# B&R Automation Studio project OpcUaSample410_BrbLibUa103 (part 9)

#### Types.typ - Exported data types
```iecst
(*General*)

TYPE
	BrbErrorUa_ENUM :
		( (*OpcUa-Error-Stati*)
		eBRB_ERR_UA_ERROR := 51000,
		eBRB_ERR_UA_NO_ELEMENTS := 51001,
		eBRB_ERR_UA_INVALID_INDEX := 51002,
		eBRB_ERR_UA_NOT_CONNECTED := 51003,
		eBRB_ERR_UA_NOT_RUNNING := 51004
		);
END_TYPE

(*General - Attributes*)

TYPE
	BrbUaNodeInfoAttribute_TYP : 	STRUCT  (*Attribut-Info*)
		sName : STRING[nBRBUA_ATTRIBUTE_NAME_CHAR_MAX]; (*Name des Attributs*)
		sValue : STRING[nBRBUA_VALUE_TEXT_CHAR_MAX]; (*Wert des Attributs als Text*)
	END_STRUCT;
	BrbUaNodeInfoAttributes_TYP : 	STRUCT  (*Attribute-Liste der Infos*)
		Attribute : ARRAY[0..nBRBUA_ATTRIBUTES_INDEX_MAX]OF BrbUaNodeInfoAttribute_TYP; (*Attribute-Liste der Infos*)
	END_STRUCT;
END_TYPE

(*General - ByteStrings*)
(*General - ServerInfo*)

TYPE
	BrbUaServerNamespacesArray_TYP : 	STRUCT  (*Array für Namespaces*)
		Length : UAArrayLength;
		Data : ARRAY[0..nBRBUA_SRVDIAG_NAMESPACE_IDX_MAX]OF STRING[nBRBUA_NAMESPACE_URI_CHAR_MAX];
	END_STRUCT;
	BrbUaServerBuildInfo_TYP : 	STRUCT  (*Build-Daten des Servers*)
		sProductUri : STRING[255];
		sManufacturerName : STRING[255];
		sProductName : STRING[255];
		sSoftwareVersion : STRING[255];
		sBuildNumber : STRING[255];
		dtBuildDate : DATE_AND_TIME;
	END_STRUCT;
	BrbUaServerState_ENUM :
		( (*Server-Status*)
		eBRBUA_SRVSTATE_RUNNING,
		eBRBUA_SRVSTATE_FAILED,
		eBRBUA_SRVSTATE_NOCONFIG,
		eBRBUA_SRVSTATE_SUSPENDED,
		eBRBUA_SRVSTATE_SHUTDOWN,
		eBRBUA_SRVSTATE_TEST,
		eBRBUA_SRVSTATE_COMMFAULT,
		eBRBUA_SRVSTATE_UNKNOWN
		);
	BrbUaServerStatus_TYP : 	STRUCT  (*Status-Daten des Servers*)
		dtStartTime : DATE_AND_TIME;
		dtCurrentTime : DATE_AND_TIME;
		eServerState : BrbUaServerState_ENUM;
		BuildInfo : BrbUaServerBuildInfo_TYP;
		nSecondsTillShutdown : UDINT;
		ShutdownReason : UALocalizedText;
	END_STRUCT;
END_TYPE

(*General - ServerDiag*)

TYPE
	BrbUaServerDiagData_TYP : 	STRUCT  (*Diagnose-Daten einer Session*)
		nServerViewCount : UDINT;
		nCurrentSessionCount : UDINT;
		nCumulatedSessionCount : UDINT;
		nSecurityRejectedSessionCount : UDINT;
		nRejectedSessionCount : UDINT;
		nSessionTimeoutCount : UDINT;
		nSessionAbortCount : UDINT;
		nCurrentSubscriptionCount : UDINT;
		nCumulatedSubscriptionCount : UDINT;
		nPublishingIntervalCount : UDINT;
		nSecurityRejectedRequestsCount : UDINT;
		nRejectedRequestsCount : UDINT;
	END_STRUCT;
	BrbUaApplicationType_ENUM :
		( (*Applikations-Typen*)
		eBRBUA_APPTYPE_SERVER, (*Nur Server*)
		eBRBUA_APPTYPE_CLIENT, (*Nur Client*)
		eBRBUA_APPTYPE_CLIENT_AND_SERVER, (*Client und Server*)
		eBRBUA_APPTYPE_DISCOVERY_SERVER (*Nur Discovery-Server*)
		);
	BrbUaApplicationDescription_TYP : 	STRUCT  (*Applikations-Beschreibung*)
		sApplicationUri : STRING[255];
		sProductUri : STRING[255];
		ApplicationName : UALocalizedText;
		eApplicationType : BrbUaApplicationType_ENUM;
		sGatewayServerUri : STRING[255];
		sDiscoveryProfileUri : STRING[255];
		DiscoveryUrlsLength : UANoOfElements;
		sDiscoveryUrls : ARRAY[0..9]OF STRING[255];
	END_STRUCT;
	BrbUaServiceCounterData_TYP : 	STRUCT  (*Zähler für Service-Daten*)
		nTotalCount : UDINT;
		nErrorCount : UDINT;
	END_STRUCT;
	BrbUaSessDiagData_TYP : 	STRUCT  (*Diagnose-Daten einer Session*)
		SessionId : UANodeID;
		sSessionName : STRING[255];
		ClientDescription : BrbUaApplicationDescription_TYP;
		sServerUri : STRING[255];
		sEndpointUrl : STRING[255];
		LocaleIdsCount : UANoOfElements;
		sLocaleIds : ARRAY[0..nBRBUA_SRVDIAG_LOCALES_INDEX_MAX]OF STRING[7];
		rActualSessionTimeout : LREAL;
		nMaxResponseMessageSize : UDINT;
		dtClientConnectionTime : DATE_AND_TIME;
		dtClientLastContactTime : DATE_AND_TIME;
		nCurrentSubscriptionsCount : UDINT;
		nCurrentMonitoredItemsCount : UDINT;
		nCurrentPublishRequestsInQueue : UDINT;
		TotalRequestCount : BrbUaServiceCounterData_TYP;
		nUnauthorizedRequestCount : UDINT;
		ReadCount : BrbUaServiceCounterData_TYP;
		HistoryReadCount : BrbUaServiceCounterData_TYP;
		WriteCount : BrbUaServiceCounterData_TYP;
		HistoryUpdateCount : BrbUaServiceCounterData_TYP;
		CallCount : BrbUaServiceCounterData_TYP;
		CreateMonitoredItemsCount : BrbUaServiceCounterData_TYP;
		ModifyMonitoredItemsCount : BrbUaServiceCounterData_TYP;
		SetMonitoringModeCount : BrbUaServiceCounterData_TYP;
		SetTriggeringCount : BrbUaServiceCounterData_TYP;
		DeleteMonitoredItemsCount : BrbUaServiceCounterData_TYP;
		CreateSubscriptionCount : BrbUaServiceCounterData_TYP;
		ModifySubscriptionCount : BrbUaServiceCounterData_TYP;
		SetPublishingModeCount : BrbUaServiceCounterData_TYP;
		PublishCount : BrbUaServiceCounterData_TYP;
		RepublishCount : BrbUaServiceCounterData_TYP;
		TransferSubscriptionsCount : BrbUaServiceCounterData_TYP;
		DeleteSubscriptionsCount : BrbUaServiceCounterData_TYP;
		AddNodesCount : BrbUaServiceCounterData_TYP;
		AddReferencesCount : BrbUaServiceCounterData_TYP;
		DeleteNodesCount : BrbUaServiceCounterData_TYP;
		DeleteReferencesCount : BrbUaServiceCounterData_TYP;
		BrowseCount : BrbUaServiceCounterData_TYP;
		BrowseNextCount : BrbUaServiceCounterData_TYP;
		TranslateBrowsePathToNodeIdCount : BrbUaServiceCounterData_TYP;
		QueryFirstCount : BrbUaServiceCounterData_TYP;
		QueryNextCount : BrbUaServiceCounterData_TYP;
		RegisterNodesCount : BrbUaServiceCounterData_TYP;
		UnregisterNodesCount : BrbUaServiceCounterData_TYP;
	END_STRUCT;
	BrbUaSessDiagArray_TYP : 	STRUCT  (*Array für Session-Diagnose*)
		Length : UAArrayLength;
		Data : ARRAY[0..nBRBUA_SRVDIAG_SESSION_INDEX_MAX]OF BrbUaSessDiagData_TYP;
	END_STRUCT;
	BrbUaMessageSecurityMode_ENUM :
		( (*Message-Secutity-Modes*)
		eBRBUA_SECMODE_INVALID, (*Ungültig*)
		eBRBUA_SECMODE_NONE, (*Keine Security*)
		eBRBUA_SECMODE_SIGN, (*Nur Signierung*)
		eBRBUA_SECMODE_SIGN_AND_ENCRYPT (*Signierung und Verschlüsselung*)
		);
	BrbUaSessSecDiagData_TYP : 	STRUCT  (*Security-Diagnose-Daten einer Session*)
		SessionId : UANodeID;
		sClientUserIdOfSession : STRING[64];
		ClientUserIdHistoryCount : UANoOfElements;
		sClientUserIdHistory : ARRAY[0..nBRBUA_SRVDIAG_USERHIST_IDX_MAX]OF STRING[32];
		sAuthenticationMechanism : STRING[64];
		sEncoding : STRING[64];
		sTransportProtocol : STRING[64];
		eSecurityMode : BrbUaMessageSecurityMode_ENUM;
		sSecurityPolicyUri : STRING[64];
		ClientCertificate : ARRAY[0..nBRBUA_CERT_ARRAY_INDEX_MAX]OF USINT;
	END_STRUCT;
	BrbUaSessSecDiagArray_TYP : 	STRUCT  (*Array für Security-Session-Diagnose*)
		Length : UAArrayLength;
		Data : ARRAY[0..nBRBUA_SRVDIAG_SESSION_INDEX_MAX]OF BrbUaSessSecDiagData_TYP;
	END_STRUCT;
	BrbUaSubscriptDiagData_TYP : 	STRUCT  (*Diagnose-Daten einer Subscription*)
		SessionId : UANodeID;
		nSubscriptionId : UDINT;
		nPriority : USINT;
		rPublishingInterval : LREAL;
		nMaxKeepAliveCount : UDINT;
		nMaxLifetimeCount : UDINT;
		nMaxNotificationsPerPublish : UDINT;
		bPublishingEnabled : BOOL;
		nModifyCount : UDINT;
		nEnableCount : UDINT;
		nDisableCount : UDINT;
		nRepublishRequestCount : UDINT;
		nRepublishMessageRequestCount : UDINT;
		nRepublishMessageCount : UDINT;
		nTransferRequestCount : UDINT;
		nTransferredToAltClientCount : UDINT;
		nTransferredToSameClientCount : UDINT;
		nPublishRequestCount : UDINT;
		nDataChangeNotificationsCount : UDINT;
		nEventNotificationsCount : UDINT;
		nNotificationsCount : UDINT;
		nLatePublishRequestCount : UDINT;
		nCurrentKeepAliveCount : UDINT;
		nCurrentLifetimeCount : UDINT;
		nUnacknowledgedMessageCount : UDINT;
		nDiscardedMessageCount : UDINT;
		nMonitoredItemCount : UDINT;
		nDisabledMonitoredItemCount : UDINT;
		nMonitoringQueueOverflowCount : UDINT;
		nNextSequenceNumber : UDINT;
		nEventQueueOverflowCount : UDINT;
	END_STRUCT;
	BrbUaSubscriptDiagArray_TYP : 	STRUCT  (*Array für Subscription-Diagnose*)
		Length : UAArrayLength;
		Data : ARRAY[0..nBRBUA_SRVDIAG_SUBSCR_INDEX_MAX]OF BrbUaSubscriptDiagData_TYP;
	END_STRUCT;
END_TYPE

(*Client - RunClient*)

TYPE
	UAByteStringBrbEventId_TYP : 	STRUCT  (*EventId als ByteString mit Länge 16*)
		Length : DINT; (*Länge der Daten (sollte mit 16 besetzt werden)*)
		Data : ARRAY[0..nBRBUA_EVENTID_INDEX_MAX]OF USINT; (*Bytes der EventId*)
	END_STRUCT;
	BrbUaRcCfg_TYP : 	STRUCT  (*Verbindungs-Parameter*)
		sCfgDataObjName : STRING[nBRBUA_DATOBJECT_NAME_CHAR_MAX]; (*Name des Datenobjekts*)
		sServerEndpointUrl : STRING[sBRBUA_ENDPOINT_URL_CHAR_MAX]; (*Endpoint-Url*)
		SessionConnectInfo : UASessionConnectInfo; (*Angaben zur Verbindung*)
		tConnectTimeout : TIME; (*Timeout für den Connect in [ms]*)
		tAccessTimeout : TIME; (*Timeout für Zugriff auf den Server in [ms]*)
	END_STRUCT;
	BrbUaRcCommandos_ENUM :
		( (*Client-Kommandos*)
		eBRB_RCCLTCMD_NONE, (*Aktuell kein Kommando*)
		eBRB_RCCLTCMD_CONNECT, (*Verbindung aufbauen*)
		eBRB_RCCLTCMD_DISCONNECT (*Verbindung trennen*)
		);
	BrbUaRcConnection_TYP : 	STRUCT  (*Daten der Verbindung*)
		nConnectionHandle : UDINT; (*Handle der Verbindung*)
		nErrorId : DWORD; (*OpcUa-Fehler beim Verbinden*)
		nConnectTries : UDINT; (*Connect-Versuche*)
		nInterruptedCount : UDINT; (*Anzahl der Verbindungs-Unterbrechungen*)
	END_STRUCT;
	BrbUaRcNamespaces_TYP : 	STRUCT  (*Daten der Namespaces*)
		nNamespaceCount : UINT; (*Anzahl der Namespaces*)
		pNamespaces : {REDUND_UNREPLICABLE} UDINT; (*Interner Zeiger*)
		nMemLen : UDINT; (*Interne Speichergröße*)
	END_STRUCT;
	BrbUaRcNamespace_TYP : 	STRUCT  (*Daten eines Namespaces*)
		sNamespaceUri : STRING[nBRBUA_NAMESPACE_URI_CHAR_MAX]; (*Namespace-Uri aus dem Datenobjekt*)
		nNamespaceIndex : UINT; (*Server-Namespace-Index*)
		nErrorId : DWORD; (*OpcUa-Fehler-Status*)
	END_STRUCT;
	BrbUaRcNodeHandles_TYP : 	STRUCT  (*Daten der NodeHandles*)
		nNodeHandleCount : UINT; (*Anzahl der NodeHandles*)
		pStart : UDINT; (*Interner Zeiger*)
		pDatObjNamespaceIndices : {REDUND_UNREPLICABLE} UDINT; (*Interner Zeiger*)
		pNodeIds : {REDUND_UNREPLICABLE} UDINT; (*Interner Zeiger*)
		pNodeHandleErrorIds : {REDUND_UNREPLICABLE} UDINT; (*Interner Zeiger*)
		pNodeHandles : {REDUND_UNREPLICABLE} UDINT; (*Interner Zeiger*)
		nMemLen : UDINT; (*Interne Speichergröße*)
	END_STRUCT;
	BrbUaRcNodeHandle_TYP : 	STRUCT  (*Daten eines NodeHandles*)
		nDatObjNamespaceIndex : UINT; (*Namespace-Index laut Datenobjekt*)
		NodeId : UANodeID; (*NodeId laut Datenobjekt*)
		nErrorId : DWORD; (*OpcUa-Fehler-Status beim Ermitteln des NodeHandles*)
		nNodeHandle : DWORD; (*Ermittelter NodeHandle*)
	END_STRUCT;
	BrbUaRcReadBlocks_TYP : 	STRUCT  (*Daten der ReadBlocks*)
		nBlockCount : UINT; (*Anzahl der ReadBlocks*)
		pBlocks : {REDUND_UNREPLICABLE} UDINT; (*Interner Zeiger*)
		nMemLen : UDINT; (*Interne Speichergröße*)
	END_STRUCT;
	BrbUaRcReadBlockIntern_TYP : 	STRUCT  (*Interne Daten eines ReadBlocks*)
		nReadItemCount : UINT; (*Anzahl der ReadItems*)
		pRiStart : UDINT; (*Interner Zeiger*)
		pRiDatObjNamespaceIndices : UDINT; (*Interner Zeiger*)
		pRiNodeIds : UDINT; (*Interner Zeiger*)
		pRiNodeAddInfos : UDINT; (*Interner Zeiger*)
		pRiVariables : UDINT; (*Interner Zeiger*)
		pRiNodeErrorIds : UDINT; (*Interner Zeiger*)
		pRiTimestamps : UDINT; (*Interner Zeiger*)
		nMemLen : UDINT; (*Interne Speichergröße*)
	END_STRUCT;
	BrbUaRcReadBlock_TYP : 	STRUCT  (*Daten eines ReadBlocks*)
		nReadItemCount : UINT; (*Anzahl der ReadItems*)
	END_STRUCT;
	BrbUaRcReadItem_TYP : 	STRUCT  (*Daten eines ReadItems*)
		nDatObjNamespaceIndex : UINT; (*Namespace-Index laut Datenobjekt*)
		NodeId : UANodeID; (*NodeId laut Datenobjekt*)
		AddInfo : UANodeAdditionalInfo; (*Zusatzangaben für den Zugriff*)
		sVar : STRING[nBRBUA_VARNAME_TEXT_CHAR_MAX]; (*Name der gemappten Variable*)
		dtTimestamp : DATE_AND_TIME; (*Zeitstempel der letzten Aktion*)
		nErrorId : DWORD; (*OpcUa-Fehler-Status*)
	END_STRUCT;
	BrbUaRcWriteBlocks_TYP : 	STRUCT  (*Daten der WriteBlocks*)
		nBlockCount : UINT; (*Anzahl der WriteBlocks*)
		pBlocks : {REDUND_UNREPLICABLE} UDINT; (*Interner Zeiger*)
		nMemLen : UDINT; (*Interne Speichergröße*)
	END_STRUCT;
	BrbUaRcWriteBlockIntern_TYP : 	STRUCT  (*Interne Daten eines WriteBlocks*)
		nWriteItemCount : UINT; (*Anzahl der WriteBlocks*)
		pWiStart : UDINT; (*Interner Zeiger*)
		pWiDatObjNamespaceIndices : UDINT; (*Interner Zeiger*)
		pWiNodeIds : UDINT; (*Interner Zeiger*)
		pWiNodeAddInfos : UDINT; (*Interner Zeiger*)
		pWiVariables : UDINT; (*Interner Zeiger*)
		pWiNodeErrorIds : UDINT; (*Interner Zeiger*)
		nMemLen : UDINT; (*Interne Speichergröße*)
	END_STRUCT;
	BrbUaRcWriteBlock_TYP : 	STRUCT  (*Daten eines WriteBlocks*)
		nWriteItemCount : UINT; (*Anzahl der WriteItems*)
	END_STRUCT;
	BrbUaRcWriteItem_TYP : 	STRUCT  (*Daten eines WriteItems*)
		nDatObjNamespaceIndex : UINT; (*Namespace-Index laut Datenobjekt*)
		NodeId : UANodeID; (*NodeId laut Datenobjekt*)
		AddInfo : UANodeAdditionalInfo; (*Zusatzangaben für den Zugriff*)
		sVar : STRING[nBRBUA_VARNAME_TEXT_CHAR_MAX]; (*Name der gemappten Variable*)
		nErrorId : DWORD; (*OpcUa-Fehler-Status*)
	END_STRUCT;
	BrbUaRcMethods_TYP : 	STRUCT  (*Daten der Methods*)
		nMethodCount : UINT; (*Anzahl der Methods*)
		pMethods : {REDUND_UNREPLICABLE} UDINT; (*Interner Zeiger*)
		nMemLen : UDINT; (*Interne Speichergröße*)
	END_STRUCT;
	BrbUaRcMethodIntern_TYP : 	STRUCT  (*Interne Daten einer Method*)
		nDatObjNamespaceIndex : UINT; (*Namespace-Index laut Datenobjekt*)
		ObjectNodeId : UANodeID; (*NodeId laut Datenobjekt*)
		MethodNodeId : UANodeID; (*NodeId laut Datenobjekt*)
		tTimeout : TIME; (*Timeout für den Call*)
		pStart : UDINT; (*Interner Zeiger*)
		nInputArgsCount : USINT; (*Anzahl der Eingangs-Argumente*)
		pInputArguments : UDINT; (*Interner Zeiger*)
		nOutputArgsCount : USINT; (*Anzahl der Ausgangs-Argumente*)
		pOutputArguments : UDINT; (*Interner Zeiger*)
		nMemLen : UDINT; (*Interne Speichergröße*)
		nErrorId : DWORD; (*OpcUa-Fehler-Status beim Ermitteln des MethodHandles*)
		nMethodHandle : DWORD; (*Ermittelter MethodHandle*)
	END_STRUCT;
	BrbUaRcMethod_TYP : 	STRUCT  (*Daten einer Method*)
		nDatObjNamespaceIndex : UINT; (*Namespace-Index laut Datenobjekt*)
		ObjectNodeId : UANodeID; (*NodeId laut Datenobjekt*)
		MethodNodeId : UANodeID; (*NodeId laut Datenobjekt*)
		tTimeout : TIME; (*Timeout für den Call*)
		nInputArgsCount : USINT; (*Anzahl der Eingangs-Argumente*)
		nOutputArgsCount : USINT; (*Anzahl der Ausgangs-Argumente*)
		nErrorId : DWORD; (*OpcUa-Fehler-Status beim Ermitteln des MethodHandles*)
		nMethodHandle : DWORD; (*Ermittelter MethodHandle*)
	END_STRUCT;
	BrbUaRcSubscriptions_TYP : 	STRUCT  (*Daten der Subscriptions*)
		nSubscriptionCount : UINT; (*Anzahl der Subscriptions*)
		pSubscriptions : {REDUND_UNREPLICABLE} UDINT; (*Interner Zeiger*)
		nMemLen : UDINT; (*Interne Speichergröße*)
		nMonitoredItemsCountTotal : UDINT; (*Anzahl aller MonitorredItems*)
		nEventItemsCountTotal : UDINT; (*Anzahl aller EventItems*)
	END_STRUCT;
	BrbUaRcSubscriptionIntern_TYP : 	STRUCT  (*Interne Daten einer Subscription*)
		bPublishingEnable : BOOL; (*Aktivierung der Subscription*)
		nPriority : USINT; (*Priorität (0..255, je größer desto höher)*)
		tPublishingInterval : TIME; (*Sende-Intervall in [ms]*)
		nMonitoredItemCount : UINT; (*Anzahl der MonitoredItems*)
		nEventItemCount : UINT; (*Anzahl der EventItems*)
		nErrorId : DWORD; (*OpcUa-Fehler-Status*)
		nSubscriptionHandle : DWORD; (*Ermitteltes SubscriptionHandle*)
		pMiStart : UDINT; (*Interner Zeiger*)
		pMiDatObjNamespaceIndices : UDINT; (*Interner Zeiger*)
		pMiNodeIds : UDINT; (*Interner Zeiger*)
		pMiNodeHandleErrorIds : UDINT; (*Interner Zeiger*)
		pMiNodeHandles : UDINT; (*Interner Zeiger*)
		pMiNodeAddInfos : UDINT; (*Interner Zeiger*)
		pMiVariables : UDINT; (*Interner Zeiger*)
		pMiQueueSizeOri : UDINT; (*Interner Zeiger*)
		pMiMonitorSettings : UDINT; (*Interner Zeiger*)
		pMiValuesChanged : UDINT; (*Interner Zeiger*)
		pMiRemainingValueCounts : UDINT; (*Interner Zeiger*)
		pMiTimestamps : UDINT; (*Interner Zeiger*)
		pMiNodeQualityIds : UDINT; (*Interner Zeiger*)
		pMiMonitoredItemErrorIds : UDINT; (*Interner Zeiger*)
		pMiMonitoredItemHandles : UDINT; (*Interner Zeiger*)
		nMiMemLen : UDINT; (*Interne Speichergröße*)
		pEventItems : UDINT; (*Interner Zeiger*)
		nEiMemLen : UDINT; (*Interne Speichergröße*)
	END_STRUCT;
	BrbUaRcSubscription_TYP : 	STRUCT  (*Daten einer Subscription*)
		bPublishingEnable : BOOL; (*Aktivierung der Subscription*)
		nPriority : USINT; (*Priorität (0..255, je größer desto höher)*)
		tPublishingInterval : TIME; (*Sende-Intervall in [ms]*)
		nMonitoredItemCount : UINT; (*Anzahl der MonitoredItems*)
		nEventItemCount : UINT; (*Anzahl der EventItems*)
		nErrorId : DWORD; (*OpcUa-Fehler-Status*)
		nSubscriptionHandle : DWORD; (*Ermitteltes SubscriptionHandle*)
	END_STRUCT;
	BrbUaRcMonitoredItem_TYP : 	STRUCT  (*Daten eines MonitoredItems*)
		nDatObjNamespaceIndex : UINT; (*Namespace-Index laut Datenobjekt*)
		NodeId : UANodeID; (*NodeId laut Datenobjekt*)
		nNodeHandleErrorId : DWORD; (*OpcUa-Fehler-Status*)
		nNodeHandle : DWORD; (*Ermitteltes NodeHandle*)
		AddInfo : UANodeAdditionalInfo; (*Zusatzangaben für den Zugriff*)
		sVar : STRING[nBRBUA_VARNAME_TEXT_CHAR_MAX]; (*Name der gemappten Variable*)
		nQueueSizeOri : UINT; (*Puffergröße laut Datenobjekt*)
		MonitorSettings : UAMonitoringParameters; (*Überwachungs-Einstellungen*)
		bValueChanged : BOOL; (*1=Wert hat sich geändert*)
		nRemainingValueCount : UINT; (*Anzahl der verbleibenden Wert-Änderungen*)
		dtTimestamp : DATE_AND_TIME; (*Zeitstempel der letzten Wert-Änderung*)
		nNodeQualityId : DWORD; (*OpcUa-Fehler-Status der letzten Wert-Änderung*)
		nMonitoredItemErrorId : DWORD; (*OpcUa-Fehler-Status*)
		nMonitoredItemHandle : DWORD; (*Ermitteltes MonitoredItemHandle*)
	END_STRUCT;
	BrbUaRcEventItemIntern_TYP : 	STRUCT  (*Interne Daten eines EventItems*)
		nEventDatObjNamespaceIndex : UINT; (*Namespace-Index laut Datenobjekt*)
		EventNodeId : UANodeID; (*NodeId laut Datenobjekt*)
		nEventNodeHandleErrorId : DWORD; (*OpcUa-Fehler-Status*)
		nEventNodeHandle : DWORD; (*Ermitteltes NodeHandle*)
		nTypeDatObjNamespaceIndex : UINT; (*Namespace-Index laut Datenobjekt*)
		TypeNodeId : UANodeID; (*NodeId laut Datenobjekt*)
		nEventItemErrorId : DWORD; (*OpcUa-Fehler-Status*)
		nEventItemHandle : DWORD; (*Ermitteltes NodeHandle*)
		tTimeout : TIME; (*Timeout für Operate in [ms]*)
		bCallOperate : BOOL; (*1=Zyklischer Aufruf von Operate*)
		nEventFieldCount : UINT; (*Anzahl der Fields*)
		pEfStart : UDINT; (*Interner Zeiger*)
		pEfDatObjNamespaceIndices : UDINT; (*Interner Zeiger*)
		pEfFieldSelections : UDINT; (*Interner Zeiger*)
		pEfFieldVars : UDINT; (*Interner Zeiger*)
		nEfMemLen : UDINT; (*Interne Speichergröße*)
		nReceiveCount : UDINT; (*Empfangs-Zähler*)
		bEventReceived : BOOL; (*Empfangs-Flag*)
	END_STRUCT;
	BrbUaRcEventItem_TYP : 	STRUCT  (*Daten eines EventItems*)
		nEventDatObjNamespaceIndex : UINT; (*Namespace-Index laut Datenobjekt*)
		EventNodeId : UANodeID; (*NodeId laut Datenobjekt*)
		nEventNodeHandleErrorId : DWORD; (*OpcUa-Fehler-Status*)
		nEventNodeHandle : DWORD; (*Ermitteltes NodeHandle*)
		nTypeDatObjNamespaceIndex : UINT; (*Namespace-Index laut Datenobjekt*)
		TypeNodeId : UANodeID; (*NodeId laut Datenobjekt*)
		nEventItemErrorId : DWORD; (*OpcUa-Fehler-Status*)
		nEventItemHandle : DWORD; (*Ermitteltes NodeHandle*)
		tTimeout : TIME; (*Timeout für Operate in [ms]*)
		bCallOperate : BOOL; (*1=Zyklischer Aufruf von Operate*)
		nEventFieldCount : UINT; (*Anzahl der Fields*)
		nReceiveCount : UDINT; (*Empfangs-Zähler*)
		bEventReceived : BOOL; (*1=Event wurde empfangen (nur für einen Zyklus)*)
	END_STRUCT;
	BrbUaRcEventField_TYP : 	STRUCT  (*Daten eines EventFields*)
		nDatObjNamespaceIndex : UINT; (*Namespace-Index laut Datenobjekt*)
		FieldSelection : UARelativePath; (*Angaben zum Field*)
		sVar : STRING[nBRBUA_VARNAME_TEXT_CHAR_MAX]; (*Name der gemappten Variable*)
	END_STRUCT;
	BrbUaRcClientStates_ENUM :
		( (*Stati des RunClients*)
		eBRB_RCCLTSTATE_NO_INIT,
		eBRB_RCCLTSTATE_INITIALIZING,
		eBRB_RCCLTSTATE_INIT_ERROR,
		eBRB_RCCLTSTATE_INIT_DONE,
		eBRB_RCCLTSTATE_WAIT_FOR_CONNECT,
		eBRB_RCCLTSTATE_CONNECTING,
		eBRB_RCCLTSTATE_CONNECT_ERROR,
		eBRB_RCCLTSTATE_CON_INTERRUPTED,
		eBRB_RCCLTSTATE_CONNECTED,
		eBRB_RCCLTSTATE_DISCONNECTING,
		eBRB_RCCLTSTATE_DISCONNECT_ERROR,
		eBRB_RCCLTSTATE_DISCONNECTED,
		eBRB_RCCLTSTATE_EXITING,
		eBRB_RCCLTSTATE_EXIT_ERROR,
		eBRB_RCCLTSTATE_EXIT_DONE
		);
	BrbUaRcStateConStatus_TYP : 	STRUCT  (*Status des Servers*)
		eConnectionStatus : {REDUND_UNREPLICABLE} UAConnectionStatus; (*Status der Verbindung*)
		eServerState : UAServerState; (*Status des Servers*)
		nServiceLevel : USINT; (*Level des Servers*)
	END_STRUCT;
	BrbUaRcState_TYP : 	STRUCT  (*Status des Clients und der Verbindung und des Servers*)
		eClientState : {REDUND_UNREPLICABLE} BrbUaRcClientStates_ENUM; (*Status des Clients*)
		nClientErroId : UDINT; (*OpcUa-Fehler-Status bei internen Aufrufen*)
		sClientErrorText : STRING[nBRBUA_VALUE_TEXT_CHAR_MAX]; (*Details zum Fehler*)
		ConnectionStatus : BrbUaRcStateConStatus_TYP; (*Status des Servers*)
	END_STRUCT;
	BrbUaRunClient_TYP : 	STRUCT  (*RunClient-Struktur zum Betreiben eines Clients*)
		Cfg : BrbUaRcCfg_TYP; (*Verbindungs-Parameter*)
		eCmd : BrbUaRcCommandos_ENUM; (*Client-Kommandos (z.B. Verbindung trennen)*)
		Connection : BrbUaRcConnection_TYP; (*Daten der Verbindung*)
		Namespaces : BrbUaRcNamespaces_TYP; (*Daten der Namespaces*)
		NodeHandles : BrbUaRcNodeHandles_TYP; (*Daten der NodeHandles*)
		ReadBlocks : BrbUaRcReadBlocks_TYP; (*Daten der ReadBlocks*)
		WriteBlocks : BrbUaRcWriteBlocks_TYP; (*Daten der WriteBlocks*)
		Methods : BrbUaRcMethods_TYP; (*Daten der Methods*)
		Subscriptions : BrbUaRcSubscriptions_TYP; (*Daten der Subscriptions*)
		State : BrbUaRcState_TYP; (*Status des Clients, der Verbindung und des Servers*)
	END_STRUCT;
	BrbUaRcMonitorNamespace_TYP : 	STRUCT  (*Interne Daten zu einem Namespace*)
		nDatObjNamespaceIndex : UINT; (*Namespace-Index laut Datenobjekt*)
		Namespace : BrbUaRcNamespace_TYP; (*Daten des Namespaces*)
	END_STRUCT;
	BrbUaRcMonitorNodeHandle_TYP : 	STRUCT  (*Interne Daten zu einem NodeHandle*)
		nNodeHandleIndex : UINT; (*0-basierter Index des NodeHandles*)
		nMonitorStatus : UINT; (*Status des Monitors*)
		NodeHandle : BrbUaRcNodeHandle_TYP; (*Daten des NodeHandles*)
	END_STRUCT;
	BrbUaRcMonitorReadBlock_TYP : 	STRUCT  (*Interne Daten zu einem ReadBlock*)
		nReadBlockIndex : UINT; (*0-basierter Index des ReadBlocks*)
		nMonitorStatus : UINT; (*Status des Monitors*)
		ReadBlock : BrbUaRcReadBlock_TYP; (*Daten des ReadBlocks*)
		ReadBlockIntern : BrbUaRcReadBlockIntern_TYP; (*Interne Daten des ReadBlocks*)
	END_STRUCT;
	BrbUaRcMonitorReadItem_TYP : 	STRUCT  (*Interne Daten zu einem ReadItem*)
		nReadBlockIndex : UINT; (*0-basierter Index des ReadBlocks*)
		nReadItemIndex : UINT; (*0-basierter Index des ReadItems*)
		nMonitorStatus : UINT; (*Status des Monitors*)
		ReadItem : BrbUaRcReadItem_TYP; (*Daten des ReadItems*)
	END_STRUCT;
	BrbUaRcMonitorWriteBlock_TYP : 	STRUCT  (*Interne Daten zu einem WriteBlock*)
		nWriteBlockIndex : UINT; (*0-basierter Index des WriteBlocks*)
		nMonitorStatus : UINT; (*Status des Monitors*)
		WriteBlock : BrbUaRcWriteBlock_TYP; (*Daten des WriteBlocks*)
		WriteBlockIntern : BrbUaRcWriteBlockIntern_TYP; (*Interne Daten des WriteBlocks*)
	END_STRUCT;
	BrbUaRcMonitorWriteItem_TYP : 	STRUCT  (*Interne Daten zu einem WriteItem*)
		nWriteBlockIndex : UINT; (*0-basierter Index des WriteBlocks*)
		nWriteItemIndex : UINT; (*0-basierter Index des WriteItems*)
		nMonitorStatus : UINT; (*Status des Monitors*)
		WriteItem : BrbUaRcWriteItem_TYP; (*Daten des WriteItems*)
	END_STRUCT;
	BrbUaRcMonitorMethod_TYP : 	STRUCT  (*Interne Daten zu einer Method*)
		nMethodIndex : UINT; (*0-basierter Index der Method*)
		nMonitorStatus : UINT; (*Status des Monitors*)
		Method : BrbUaRcMethod_TYP; (*Daten der Method*)
		MethodIntern : BrbUaRcMethodIntern_TYP; (*Interne Daten der Method*)
	END_STRUCT;
	BrbUaRcMonitorArgument_TYP : 	STRUCT  (*Interne Daten zu einem Argument*)
		nMethodIndex : UINT; (*0-basierter Index der Method*)
		bOutput : BOOL; (*0=Eingangs-Argument, 1=Ausgangs-Argument*)
		nArgumentIndex : UINT; (*0-basierter Index des Arguments*)
		nMonitorStatus : UINT; (*Status des Monitors*)
		Argument : UAMethodArgument; (*Daten des Arguments*)
	END_STRUCT;
	BrbUaRcMonitorSubscription_TYP : 	STRUCT  (*Interne Daten zu einer Subscription*)
		nSubscriptionIndex : UINT; (*0-basierter Index der Subscription*)
		nMonitorStatus : UINT; (*Status des Monitors*)
		Subscription : BrbUaRcSubscription_TYP; (*Daten einer Subscription*)
		SubscriptionIntern : BrbUaRcSubscriptionIntern_TYP; (*Interne Daten der Subscription*)
	END_STRUCT;
	BrbUaRcMonitorMonitoredItem_TYP : 	STRUCT  (*Interne Daten zu einem MonitoredItem*)
		nSubscriptionIndex : UINT; (*0-basierter Index der Subscription*)
		nMonitoredItemIndex : UINT; (*0-basierter Index des MonitoredItems*)
		nMonitorStatus : UINT; (*Status des Monitors*)
		MonitoredItem : BrbUaRcMonitoredItem_TYP; (*Daten des MonitoredItems*)
	END_STRUCT;
	BrbUaRcMonitorEventItem_TYP : 	STRUCT  (*Interne Daten zu einem EventItem*)
		nSubscriptionIndex : UINT; (*0-basierter Index der Subscription*)
		nEventItemIndex : UINT; (*0-basierter Index des EventItems*)
		nMonitorStatus : UINT; (*Status des Monitors*)
		EventItem : BrbUaRcEventItem_TYP; (*Daten des EventItems*)
		EventItemIntern : BrbUaRcEventItemIntern_TYP; (*Interne Daten des EventItems*)
	END_STRUCT;
	BrbUaRcMonitorEventField_TYP : 	STRUCT  (*Interne Daten zu einem EventField*)
		nSubscriptionIndex : UINT; (*0-basierter Index der Subscription*)
		nEventItemIndex : UINT; (*0-basierter Index des EventItems*)
		nEventFieldIndex : UINT; (*0-basierter Index des EventFields*)
		nMonitorStatus : UINT; (*Status des Monitors*)
		EventField : BrbUaRcEventField_TYP; (*Daten eines EventFields*)
	END_STRUCT;
	BrbUaRcMonitor_TYP : 	STRUCT  (*Monitor für interne Daten*)
		bEnable : BOOL; (*1=Aktiv*)
		nMonitorStatus : UINT; (*Status des Monitors*)
		Namespace : BrbUaRcMonitorNamespace_TYP; (*Interne Daten zu einem Namespace*)
		NodeHandle : BrbUaRcMonitorNodeHandle_TYP; (*Interne Daten zu einem NodeHandle*)
		ReadBlock : BrbUaRcMonitorReadBlock_TYP; (*Interne Daten zu einem ReadBlock*)
		ReadItem : BrbUaRcMonitorReadItem_TYP; (*Interne Daten zu einem ReadItem*)
		WriteBlock : BrbUaRcMonitorWriteBlock_TYP; (*Interne Daten zu einem WriteBlock*)
		WriteItem : BrbUaRcMonitorWriteItem_TYP; (*Interne Daten zu einem WriteItem*)
		Method : BrbUaRcMonitorMethod_TYP; (*Interne Daten zu einer Method*)
		Argument : BrbUaRcMonitorArgument_TYP; (*Interne Daten zu einem Argument*)
		Subscription : BrbUaRcMonitorSubscription_TYP; (*Interne Daten zu einer Subscription*)
		MonitoredItem : BrbUaRcMonitorMonitoredItem_TYP; (*Interne Daten zu einem MonitoredItem*)
		EventItem : BrbUaRcMonitorEventItem_TYP; (*Interne Daten zu einem EventItem*)
		EventField : BrbUaRcMonitorEventField_TYP; (*Interne Daten zu einem EventField*)
	END_STRUCT;
END_TYPE

(*Server - Methods*)

TYPE
	BrbUaSrvMethodPar_TYP : 	STRUCT  (*Parameter einer Methode*)
		sMethodName : STRING[nBRBUA_METHOD_CHAR_MAX]; (*Name der Methode*)
		bEnable : BOOL; (*0=Ausführung beenden, 1=Ausführen*)
		bUserCodeIsFinished : BOOL; (*Rückmeldung, dass Benutzer-Code ausgeführt wurde*)
	END_STRUCT;
	BrbUaSrvMethodState_TYP : 	STRUCT  (*Status einer Methode*)
		bExecuteUserCode : BOOL; (*Meldung, dass Benutzer-Code ausgeführt werden muss*)
		bExecuteUserCodeInit : BOOL; (*Wird nur im ersten Zyklus gesetzt*)
		nCallCount : UINT; (*Aufruf-Zähler*)
		nErrorCount : UDINT; (*Fehler-Zähler*)
		nLastErrorId : UDINT; (*Letzter aufgetretener Fehler*)
		sLastErrorId : STRING[nBRBUA_VALUE_TEXT_CHAR_MAX]; (*Letzter aufgetretener Fehler als Hex*)
		eLastErrorAction : UaMethodOperateAction; (*Aktion beim letzten aufgetretenen Fehler*)
	END_STRUCT;
	BrbUaSrvMethodIntern_TYP : 	STRUCT  (*Intern verwendet*)
		bEnabled : BOOL; (*Interne Variable*)
		nStep : UINT; (*Step-Nummer für die interne Schrittkette*)
		fbUaSrv_MethodOperate : UaSrv_MethodOperate; (*Interner FB*)
		nErrorId : UDINT; (*Interne Variable*)
	END_STRUCT;
	BrbUaSrvMethod_TYP : 	STRUCT  (*Methode*)
		Par : BrbUaSrvMethodPar_TYP; (*Parameter*)
		State : BrbUaSrvMethodState_TYP; (*Status*)
		Intern : BrbUaSrvMethodIntern_TYP; (*Interne Variablen*)
	END_STRUCT;
END_TYPE

(*Server -RunServer*)

TYPE
	BrbUaRsCfg_TYP : 	STRUCT  (*Parameter*)
		sCfgDataObjName : STRING[nBRBUA_DATOBJECT_NAME_CHAR_MAX]; (*Name des Datenobjekts*)
	END_STRUCT;
	BrbUaRsNamespaces_TYP : 	STRUCT  (*Daten der Namespaces*)
		nNamespaceCount : UINT; (*Anzahl der Namespaces*)
		pNamespaces : {REDUND_UNREPLICABLE} UDINT; (*Interner Zeiger*)
		nMemLen : UDINT; (*Interne Speichergröße*)
	END_STRUCT;
	BrbUaRsNamespace_TYP : 	STRUCT  (*Daten eines Namespaces*)
		sNamespaceUri : STRING[nBRBUA_NAMESPACE_URI_CHAR_MAX]; (*Namespace-Uri aus dem Datenobjekt*)
		nNamespaceIndex : UINT; (*Server-Namespace-Index*)
		nErrorId : DWORD; (*OpcUa-Fehler-Status*)
	END_STRUCT;
	BrbUaRsEvents_TYP : 	STRUCT  (*Daten der Events*)
		nEventCount : UINT; (*Anzahl der Subscriptions*)
		pEvents : {REDUND_UNREPLICABLE} UDINT; (*Interner Zeiger*)
		nMemLen : UDINT; (*Interne Speichergröße*)
		nFieldsCountTotal : UDINT; (*Anzahl aller Fields aller Events*)
	END_STRUCT;
	BrbUaRsEvent_TYP : 	STRUCT  (*Daten eines Events*)
		nDatObjNamespaceIndex : UINT; (*Namespace-Index laut Datenobjekt*)
		TypeNodeId : UANodeID; (*TypeNodeId laut Datenobjekt*)
		nFieldCount : UINT; (*Anzahl der Fields*)
	END_STRUCT;
	BrbUaRsEventIntern_TYP : 	STRUCT  (*Interne Daten eines Events*)
		nDatObjNamespaceIndex : UINT; (*Namespace-Index laut Datenobjekt*)
		TypeNodeId : UANodeID; (*TypeNodeId laut Datenobjekt*)
		nFieldCount : UINT; (*Anzahl der Fields*)
		pFields : UDINT; (*Interner Zeiger*)
		nMemLen : UDINT; (*Interne Speichergröße*)
	END_STRUCT;
	BrbUaRsStates_ENUM :
		( (*Stati des RunServers*)
		eBRB_RSSTATE_NO_INIT,
		eBRB_RSSTATE_INITIALIZING,
		eBRB_RSSTATE_INIT_ERROR,
		eBRB_RSSTATE_INIT_DONE,
		eBRB_RSSTATE_DETECTING,
		eBRB_RSSTATE_RUNNING,
		eBRB_RSSTATE_EXITING,
		eBRB_RSSTATE_EXIT_ERROR,
		eBRB_RSSTATE_EXIT_DONE
		);
	BrbUaRsState_TYP : 	STRUCT  (*Status des Clients und der Verbindung und des Servers*)
		eState : {REDUND_UNREPLICABLE} BrbUaRsStates_ENUM; (*Status des RunServers*)
		nErroId : UDINT; (*OpcUa-Fehler-Status bei internen Aufrufen*)
		sErrorText : STRING[nBRBUA_VALUE_TEXT_CHAR_MAX]; (*Details zum Fehler*)
		eServerState : {REDUND_UNREPLICABLE} UAServerState; (*Status des Servers*)
	END_STRUCT;
	BrbUaRunServer_TYP : 	STRUCT  (*RunServer-Struktur zum Betreiben des RunServers*)
		Cfg : BrbUaRsCfg_TYP; (*Parameter*)
		Namespaces : BrbUaRsNamespaces_TYP; (*Daten der Namespaces*)
		Events : BrbUaRsEvents_TYP; (*Daten der Events*)
		State : BrbUaRsState_TYP; (*Status des RunServers*)
	END_STRUCT;
	BrbUaRsMonitorNamespace_TYP : 	STRUCT  (*Interne Daten zu einem Namespace*)
		nDatObjNamespaceIndex : UINT; (*Namespace-Index laut Datenobjekt*)
		Namespace : BrbUaRsNamespace_TYP; (*Daten des Namespaces*)
	END_STRUCT;
	BrbUaRsMonitorEvent_TYP : 	STRUCT  (*Interne Daten zu einer Subscription*)
		nEventIndex : UINT; (*0-basierter Index des Events*)
		nMonitorStatus : UINT; (*Status des Monitors*)
		Event : BrbUaRsEvent_TYP; (*Daten eines Events*)
		EventIntern : BrbUaRsEventIntern_TYP; (*Interne Daten eines Events*)
	END_STRUCT;
	BrbUaRsMonitorEventField_TYP : 	STRUCT  (*Interne Daten zu einem EventField*)
		nEventIndex : UINT; (*0-basierter Index des Events*)
		nEventFieldIndex : UINT; (*0-basierter Index des Fields*)
		nMonitorStatus : UINT; (*Status des Monitors*)
		Field : UaSrv_FireEventFieldType; (*Daten des Fields*)
	END_STRUCT;
	BrbUaRsMonitor_TYP : 	STRUCT  (*Monitor für interne Daten*)
		bEnable : BOOL; (*1=Aktiv*)
		nMonitorStatus : UINT; (*Status des Monitors*)
		Namespace : BrbUaRsMonitorNamespace_TYP; (*Interne Daten zu einem Namespace*)
		Event : BrbUaRsMonitorEvent_TYP; (*Interne Daten zu einem Event*)
		EventField : BrbUaRsMonitorEventField_TYP; (*Interne Daten zu einem Field*)
	END_STRUCT;
END_TYPE
```

#### Constants.var - Exported constants
```iecst
(*General*)
VAR CONSTANT
	nBRBUA_DATOBJECT_NAME_CHAR_MAX : UINT := 10; (*Anzahl der Zeichen eines Daten-Objekt-Namens*)
	sBRBUA_ENDPOINT_URL_CHAR_MAX : UINT := 255;
	nBRBUA_NAMESPACE_URI_CHAR_MAX : UINT := 255; (*Anzahl der Zeichen einer Namespace-Uri*)
	nBRBUA_CERT_NAME_CHAR_MAX : UINT := 255; (*Anzahl der Zeichen eines Variablen-Namens*)
	nBRBUA_IDENTIFIER_TEXT_CHAR_MAX : UINT := 255; (*Anzahl der Zeichen eines Identifier-Textes*)
	nBRBUA_VARNAME_TEXT_CHAR_MAX : UINT := 255; (*Anzahl der Zeichen eines Variablen-Namens*)
	nBRBUA_VALUE_TEXT_CHAR_MAX : UINT := 255; (*Anzahl der Zeichen eines Value-Textes*)
	nBRBUA_STATUS_TEXT_CHAR_MAX : UINT := 96; (*Anzahl der Zeichen eines Status-Textes*)
	nBRBUA_CERT_ARRAY_INDEX_MAX : UINT := 1999; (*Maximaler Index eines Byte-Arrays für ein Zertifikat*)
END_VAR
(*General - Attributes*)
VAR CONSTANT
	nBRBUA_ATTRIBUTE_NAME_CHAR_MAX : UINT := 32; (*Anzahl der Zeichen eines Attribut-Namens*)
	nBRBUA_ATTRIBUTES_INDEX_MAX : UINT := 22; (*Max. Index der Attribut-Liste*)
END_VAR
(*General - VariantValues*)
VAR CONSTANT
	sBRBUA_DATETIME_FORMAT : STRING[32] := 'yyyy-mm-dd hh:MM:ss'; (*Umwandlungsformat für DateTime*)
	sBRBUA_TIMESTAMP_FORMAT : STRING[nBRB_TIME_TEXT_CHAR_MAX] := 'yyyy-mm-dd hh:MM:ss'; (*Format zum Wandeln eines Zeistempels in einen Text*)
END_VAR
(*General - ByteStrings*)
VAR CONSTANT
	nBRBUA_EVENTID_INDEX_MAX : UINT := 15; (*Maximaler Index der Bytes einer EventId*)
END_VAR
(*General - ServerDiag*)
VAR CONSTANT
	nBRBUA_SRVDIAG_NAMESPACE_IDX_MAX : UINT := 19; (*Maximaler Index des Client-Diag-Arrays*)
	nBRBUA_SRVDIAG_SESSION_INDEX_MAX : UINT := 9; (*Maximaler Index des Client-Diag-Arrays*)
	nBRBUA_SRVDIAG_LOCALES_INDEX_MAX : UINT := 4; (*Maximaler Index der Locale-Liste*)
	nBRBUA_SRVDIAG_USERHIST_IDX_MAX : UINT := 4; (*Maximaler Index der User-History*)
	nBRBUA_SRVDIAG_SUBSCR_INDEX_MAX : UINT := 29; (*Maximaler Index des Subscription-Diag-Arrays*)
END_VAR
(*Client - RunClient*)
VAR CONSTANT
	nBRBUA_NAMESPACES_INDEX_MAX : UINT := 15;
	nBRBUA_CLT_READ_LINES : UINT := 100;
	nBRBUA_SRV_READ_LINES : UINT := 100;
	nBRBUA_KEYWORD_CONNECTION : STRING[nBRBUA_VALUE_TEXT_CHAR_MAX] := '§CONNECTION:';
	nBRBUA_KEYWORD_NAMESPACE : STRING[nBRBUA_VALUE_TEXT_CHAR_MAX] := '§NAMESPACE:';
	nBRBUA_KEYWORD_NODEHANDLE : STRING[nBRBUA_VALUE_TEXT_CHAR_MAX] := '§NODEHANDLE:';
	nBRBUA_KEYWORD_READBLOCK : STRING[nBRBUA_VALUE_TEXT_CHAR_MAX] := '§READBLOCK:';
	nBRBUA_KEYWORD_READITEM : STRING[nBRBUA_VALUE_TEXT_CHAR_MAX] := '§READITEM:';
	nBRBUA_KEYWORD_WRITEBLOCK : STRING[nBRBUA_VALUE_TEXT_CHAR_MAX] := '§WRITEBLOCK:';
	nBRBUA_KEYWORD_WRITEITEM : STRING[nBRBUA_VALUE_TEXT_CHAR_MAX] := '§WRITEITEM:';
	nBRBUA_KEYWORD_METHOD : STRING[nBRBUA_VALUE_TEXT_CHAR_MAX] := '§METHOD:';
	nBRBUA_KEYWORD_METHOD_ARG_IN : STRING[nBRBUA_VALUE_TEXT_CHAR_MAX] := '§METHODARGIN:';
	nBRBUA_KEYWORD_METHOD_ARG_OUT : STRING[nBRBUA_VALUE_TEXT_CHAR_MAX] := '§METHODARGOUT:';
	nBRBUA_KEYWORD_SUBSCRIPTION : STRING[nBRBUA_VALUE_TEXT_CHAR_MAX] := '§SUBSCRIPTION:';
	nBRBUA_KEYWORD_MONITORED_ITEM : STRING[nBRBUA_VALUE_TEXT_CHAR_MAX] := '§MONITEM:';
	nBRBUA_KEYWORD_EVENT_ITEM : STRING[nBRBUA_VALUE_TEXT_CHAR_MAX] := '§EVTITEM:';
	nBRBUA_KEYWORD_EVENT : STRING[nBRBUA_VALUE_TEXT_CHAR_MAX] := '§EVENT:';
	nBRBUA_KEYWORD_EVENT_FIELD : STRING[nBRBUA_VALUE_TEXT_CHAR_MAX] := '§EVTFIELD:';
END_VAR
(*Server - Methods*)
VAR CONSTANT
	nBRBUA_METHOD_CHAR_MAX : UINT := 64; (*Anzahl der Zeichen eines Methoden-Namens*)
END_VAR
```

#### AnsiCFunc.h
```c
/********************************************************************
 * COPYRIGHT -- Bernecker + Rainer
 ********************************************************************
 * Package: Global
 * File: AnsiCFunc.h
 * Author: niedermeierr
 * Created: April 22, 2008
 *******************************************************************/

#include <bur/plctypes.h>

/*
 * stdlib.h
 *
 * Definitions for common types, variables, and functions.
 */
// NOLINTBEGIN(bugprone-reserved-identifier, cert-dcl37-c, cppcoreguidelines-avoid-non-const-global-variables, clang-diagnostic-reserved-identifier)
#ifndef _STDLIB_H_
#define _STDLIB_H_

#include "_ansi.h"

#define __need_size_t
#define __need_wchar_t
#include <stddef.h>

#include <sys/reent.h>
#include <machine/stdlib.h>
#ifndef __STRICT_ANSI__
#include <alloca.h>
#endif

_BEGIN_STD_C

typedef struct
{
  int quot; /* quotient */
  int rem; /* remainder */
} div_t;

typedef struct
{
  long quot; /* quotient */
  long rem; /* remainder */
} ldiv_t;

#ifndef __STRICT_ANSI__
typedef struct
{
  long long int quot; /* quotient */
  long long int rem; /* remainder */
} lldiv_t;
#endif

#ifndef NULL
#define NULL 0
#endif

#define EXIT_FAILURE 1
#define EXIT_SUCCESS 0

#define RAND_MAX __RAND_MAX

extern __IMPORT int __mb_cur_max;

#define MB_CUR_MAX __mb_cur_max

_VOID	_EXFUN(abort,(_VOID) _ATTRIBUTE ((noreturn)));
int	_EXFUN(abs,(int));
int	_EXFUN(atexit,(_VOID (*__func)(_VOID)));
//double	_EXFUN(atof,(const char *__nptr));
#ifndef __STRICT_ANSI__
float	_EXFUN(atoff,(const char *__nptr));
#endif
//int	_EXFUN(atoi,(const char *__nptr));
int	_EXFUN(_atoi_r,(struct _reent *, const char *__nptr));
long	_EXFUN(atol,(const char *__nptr));
long	_EXFUN(_atol_r,(struct _reent *, const char *__nptr));
_PTR	_EXFUN(bsearch,(const _PTR __key,
		       const _PTR __base,
		       size_t __nmemb,
		       size_t __size,
		       int _EXPARM(_compar,(const _PTR, const _PTR))));
_PTR	_EXFUN(calloc,(size_t __nmemb, size_t __size));
div_t	_EXFUN(div,(int __numer, int __denom));
_VOID	_EXFUN(exit,(int __status) _ATTRIBUTE ((noreturn)));
_VOID	_EXFUN(free,(_PTR));
char *  _EXFUN(getenv,(const char *__string));
char *	_EXFUN(_getenv_r,(struct _reent *, const char *__string));
#ifdef __CYGWIN__
const char *_EXFUN(getprogname,(void));
#endif
char *	_EXFUN(_findenv,(_CONST char *, int *));
char *	_EXFUN(_findenv_r,(struct _reent *, _CONST char *, int *));
long	_EXFUN(labs,(long));
ldiv_t	_EXFUN(ldiv,(long __numer, long __denom));
_PTR	_EXFUN(malloc,(size_t __size));
int	_EXFUN(mblen,(const char *, size_t));
int	_EXFUN(_mblen_r,(struct _reent *, const char *, size_t, _mbstate_t *));
int	_EXFUN(mbtowc,(wchar_t *, const char *, size_t));
int	_EXFUN(_mbtowc_r,(struct _reent *, wchar_t *, const char *, size_t, _mbstate_t *));
int	_EXFUN(wctomb,(char *, wchar_t));
int	_EXFUN(_wctomb_r,(struct _reent *, char *, wchar_t, _mbstate_t *));
size_t	_EXFUN(mbstowcs,(wchar_t *, const char *, size_t));
size_t	_EXFUN(_mbstowcs_r,(struct _reent *, wchar_t *, const char *, size_t, _mbstate_t *));
size_t	_EXFUN(wcstombs,(char *, const wchar_t *, size_t));
size_t	_EXFUN(_wcstombs_r,(struct _reent *, char *, const wchar_t *, size_t, _mbstate_t *));
#ifndef __STRICT_ANSI__
#ifndef _REENT_ONLY
int     _EXFUN(mkstemp,(char *));
char *  _EXFUN(mktemp,(char *));
#endif
#endif
_VOID	_EXFUN(qsort,(_PTR __base, size_t __nmemb, size_t __size, int(*_compar)(const _PTR, const _PTR)));
int	_EXFUN(rand,(_VOID));
_PTR	_EXFUN(realloc,(_PTR __r, size_t __size));
#ifdef __CYGWIN__
void	_EXFUN(setprogname,(const char *));
#endif
_VOID	_EXFUN(srand,(unsigned __seed));
double	_EXFUN(strtod,(const char *__n, char **__end_PTR));
double	_EXFUN(_strtod_r,(struct _reent *,const char *__n, char **__end_PTR));
float	_EXFUN(strtof,(const char *__n, char **__end_PTR));
#ifndef __STRICT_ANSI__
/* the following strtodf interface is deprecated...use strtof instead */
# ifndef strtodf
#  define strtodf strtof
# endif
#endif
long	_EXFUN(strtol,(const char *__n, char **__end_PTR, int __base));
long	_EXFUN(_strtol_r,(struct _reent *,const char *__n, char **__end_PTR, int __base));
unsigned long _EXFUN(strtoul,(const char *__n, char **__end_PTR, int __base));
unsigned long _EXFUN(_strtoul_r,(struct _reent *,const char *__n, char **__end_PTR, int __base));

int	_EXFUN(system,(const char *__string));

#ifndef __STRICT_ANSI__
long    _EXFUN(a64l,(const char *__input));
char *  _EXFUN(l64a,(long __input));
char *  _EXFUN(_l64a_r,(struct _reent *,long __input));
int	_EXFUN(on_exit,(_VOID (*__func)(int, _PTR),_PTR __arg));
_VOID	_EXFUN(_Exit,(int __status) _ATTRIBUTE ((noreturn)));
int	_EXFUN(putenv,(const char *__string));
int	_EXFUN(_putenv_r,(struct _reent *, const char *__string));
int	_EXFUN(setenv,(const char *__string, const char *__value, int __overwrite));
int	_EXFUN(_setenv_r,(struct _reent *, const char *__string, const char *__value, int __overwrite));

char *	_EXFUN(gcvt,(double,int,char *));
char *	_EXFUN(gcvtf,(float,int,char *));
char *	_EXFUN(fcvt,(double,int,int *,int *));
char *	_EXFUN(fcvtf,(float,int,int *,int *));
char *	_EXFUN(ecvt,(double,int,int *,int *));
char *	_EXFUN(ecvtbuf,(double, int, int*, int*, char *));
char *	_EXFUN(fcvtbuf,(double, int, int*, int*, char *));
char *	_EXFUN(ecvtf,(float,int,int *,int *));
char *	_EXFUN(dtoa,(double, int, int, int *, int*, char**));
int	_EXFUN(rand_r,(unsigned *__seed));

double _EXFUN(drand48,(_VOID));
double _EXFUN(_drand48_r,(struct _reent *));
double _EXFUN(erand48,(unsigned short [3]));
double _EXFUN(_erand48_r,(struct _reent *, unsigned short [3]));
long   _EXFUN(jrand48,(unsigned short [3]));
long   _EXFUN(_jrand48_r,(struct _reent *, unsigned short [3]));
_VOID  _EXFUN(lcong48,(unsigned short [7]));
_VOID  _EXFUN(_lcong48_r,(struct _reent *, unsigned short [7]));
long   _EXFUN(lrand48,(_VOID));
long   _EXFUN(_lrand48_r,(struct _reent *));
long   _EXFUN(mrand48,(_VOID));
long   _EXFUN(_mrand48_r,(struct _reent *));
long   _EXFUN(nrand48,(unsigned short [3]));
long   _EXFUN(_nrand48_r,(struct _reent *, unsigned short [3]));
unsigned short *
       _EXFUN(seed48,(unsigned short [3]));
unsigned short *
       _EXFUN(_seed48_r,(struct _reent *, unsigned short [3]));
_VOID  _EXFUN(srand48,(long));
_VOID  _EXFUN(_srand48_r,(struct _reent *, long));
long long _EXFUN(atoll,(const char *__nptr));
long long _EXFUN(_atoll_r,(struct _reent *, const char *__nptr));
long long _EXFUN(llabs,(long long));
lldiv_t	_EXFUN(lldiv,(long long __numer, long long __denom));
long long _EXFUN(strtoll,(const char *__n, char **__end_PTR, int __base));
long long _EXFUN(_strtoll_r,(struct _reent *, const char *__n, char **__end_PTR, int __base));
unsigned long long _EXFUN(strtoull,(const char *__n, char **__end_PTR, int __base));
unsigned long long _EXFUN(_strtoull_r,(struct _reent *, const char *__n, char **__end_PTR, int __base));

#ifndef __CYGWIN__
_VOID	_EXFUN(cfree,(_PTR));
#else
char *	_EXFUN(realpath,(const char *, char *));
void	_EXFUN(unsetenv,(const char *__string));
void	_EXFUN(_unsetenv_r,(struct _reent *, const char *__string));
int	_EXFUN(random,(_VOID));
long	_EXFUN(srandom,(unsigned __seed));
char *  _EXFUN(ptsname, (int));
int     _EXFUN(grantpt, (int));
int     _EXFUN(unlockpt,(int));
#endif

#endif /* ! __STRICT_ANSI__ */

char *	_EXFUN(_dtoa_r,(struct _reent *, double, int, int, int *, int*, char**));
#ifndef __CYGWIN__
_PTR	_EXFUN(_malloc_r,(struct _reent *, size_t));
_PTR	_EXFUN(_calloc_r,(struct _reent *, size_t, size_t));
_VOID	_EXFUN(_free_r,(struct _reent *, _PTR));
_PTR	_EXFUN(_realloc_r,(struct _reent *, _PTR, size_t));
_VOID	_EXFUN(_mstats_r,(struct _reent *, char *));
#endif
int	_EXFUN(_system_r,(struct _reent *, const char *));

_VOID	_EXFUN(__eprintf,(const char *, const char *, unsigned int, const char *));

#ifdef __CYGWIN__
#undef _malloc_r
#define _malloc_r(r, s) malloc (s)
#undef _free_r
#define _free_r(r, p) free (p)
#undef _realloc_r
#define _realloc_r(r, p, s) realloc (p, s)
#undef _calloc_r
#define _calloc_r(r, s1, s2) calloc (s1, s2);
#undef _memalign_r
#define _memalign_r(r, s1, s2) memalign (s1, s2);
#undef _mallinfo_r
#define _mallinfo_r(r) mallinfo ()
#undef _malloc_stats_r
#define _malloc_stats_r(r) malloc_stats ()
#undef _mallopt_r
#define _mallopt_r(i1, i2) mallopt (i1, i2)
#undef _malloc_usable_size_r
#define _malloc_usable_size_r(r, p) malloc_usable_size (p)
#undef _valloc_r
#define _valloc_r(r, s) valloc (s)
#undef _pvalloc_r
#define _pvalloc_r(r, s) pvalloc (s)
#undef _malloc_trim_r
#define _malloc_trim_r(r, s) malloc_trim (s)
#undef _mstats_r
#define _mstats_r(r, p) mstats (p)
#endif

_END_STD_C

#endif /* _STDLIB_H_ */
// NOLINTEND(bugprone-reserved-identifier, cert-dcl37-c, cppcoreguidelines-avoid-non-const-global-variables, clang-diagnostic-reserved-identifier)
```

#### Package Logical/Libraries/BrbLibUa/General - Allgemeine Funktionen

#### BrbUaGetStatusCodeText.c - Gibt den symbolischen Text für einen Ua-Status-Code zurück
```c
#include <bur/plctypes.h>
#ifdef __cplusplus
	extern "C"
	{
#endif

#include "BrbLibUa.h"
#include <AnsiCFunc.h>
#include <string.h>

#ifdef __cplusplus
	};
#endif

// NOLINTBEGIN(readability-*, bugprone-easily-swappable-parameters, bugprone-branch-clone, clang-diagnostic-invalid-utf8, clang-diagnostic-invalid-source-encoding, clang-diagnostic-pointer-arith, clang-diagnostic-strict-prototypes, hicpp-uppercase-literal-suffix, cppcoreguidelines-*, performance-*)

/* Gibt den symbolischen Text für einen Ua-Status-Code zurück */
plcdword BrbUaGetStatusCodeText(unsigned long nStatusCode, plcstring* pStatusText, unsigned long nStatusTextSize)
{
	DWORD nStatus = 0x80460000; // = Bad_StructureMissing
	if(pStatusText != 0)
	{
		nStatus = 0x00000000; // = Good
		memset(pStatusText, 0, nStatusTextSize);
		BrbUdintToHex(nStatusCode, pStatusText, nStatusTextSize, 1);
		switch(nStatusCode)
		{
			case 0:
				BrbStringCat(pStatusText, " = Good", nStatusTextSize);
				break;
			case 0x002D0000:
				BrbStringCat(pStatusText, " = Good_SubscriptionTransferred", nStatusTextSize);
				break;
			case 0x002E0000:
				BrbStringCat(pStatusText, " = Good_CompletesAsynchronously", nStatusTextSize);
				break;
			case 0x002F0000:
				BrbStringCat(pStatusText, " = Good_Overload", nStatusTextSize);
				break;
			case 0x00300000:
				BrbStringCat(pStatusText, " = Good_Clamped", nStatusTextSize);
				break;
			case 0x00960000:
				BrbStringCat(pStatusText, " = Good_LocalOverride", nStatusTextSize);
				break;
			case 0x00A20000 :
				BrbStringCat(pStatusText, " = Good_EntryInserted", nStatusTextSize);
				break;
			case 0x00A30000:
				BrbStringCat(pStatusText, " = Good_EntryReplaced", nStatusTextSize);
				break;
			case 0x00A50000:
				BrbStringCat(pStatusText, " = Good_NoData", nStatusTextSize);
				break;
			case 0x00A60000:
				BrbStringCat(pStatusText, " = Good_MoreData", nStatusTextSize);
				break;
			case 0x00A70000:
				BrbStringCat(pStatusText, " = Good_CommunicationEvent", nStatusTextSize);
				break;
			case 0x00A80000:
				BrbStringCat(pStatusText, " = Good_ShutdownEvent", nStatusTextSize);
				break;
			case 0x00A90000:
				BrbStringCat(pStatusText, " = Good_CallAgain", nStatusTextSize);
				break;
			case 0x00AA0000:
				BrbStringCat(pStatusText, " = Good_NonCriticalTimeout", nStatusTextSize);
				break;
			case 0x00BA0000:
				BrbStringCat(pStatusText, " = Good_ResultsMayBeIncomplete", nStatusTextSize);
				break;
			case 0x00D90000:
				BrbStringCat(pStatusText, " = Good_DataIgnored", nStatusTextSize);
				break;

			case 0x406C0000:
				BrbStringCat(pStatusText, " = Uncertain_ReferenceOutOfServer", nStatusTextSize);
				break;
			case 0x408F0000:
				BrbStringCat(pStatusText, " = Uncertain_NoCommunicationLastUsableValue", nStatusTextSize);
				break;
			case 0x40900000:
				BrbStringCat(pStatusText, " = Uncertain_LastUsableValue", nStatusTextSize);
				break;
			case 0x40910000:
				BrbStringCat(pStatusText, " = Uncertain_SubstituteValue", nStatusTextSize);
				break;
			case 0x40920000:
				BrbStringCat(pStatusText, " = Uncertain_InitialValue", nStatusTextSize);
				break;
			case 0x40930000:
				BrbStringCat(pStatusText, " = Uncertain_SensorNotAccurate", nStatusTextSize);
				break;
			case 0x40940000:
				BrbStringCat(pStatusText, " = Uncertain_EngineeringUnitsExceeded", nStatusTextSize);
				break;
			case 0x40950000:
				BrbStringCat(pStatusText, " = Uncertain_SubNormal", nStatusTextSize);
				break;
			case 0x40A40000:
				BrbStringCat(pStatusText, " = Uncertain_DataSubNormal", nStatusTextSize);
				break;
			case 0x40BC0000:
				BrbStringCat(pStatusText, " = Uncertain_ReferenceNotDeleted", nStatusTextSize);
				break;
			case 0x40C00000:
				BrbStringCat(pStatusText, " = Uncertain_NotAllNodesAvailable", nStatusTextSize);
				break;

			case 0x80000000:
				BrbStringCat(pStatusText, " = Bad", nStatusTextSize);
				break;
			case 0x80010000:
				BrbStringCat(pStatusText, " = Bad_UnexpectedError", nStatusTextSize);
				break;
			case 0x80020000:
				BrbStringCat(pStatusText, " = Bad_InternalError", nStatusTextSize);
				break;
			case 0x80030000:
				BrbStringCat(pStatusText, " = Bad_OutOfMemory", nStatusTextSize);
				break;
			case 0x80040000:
				BrbStringCat(pStatusText, " = Bad_ResourceUnavailable", nStatusTextSize);
				break;
			case 0x80050000:
				BrbStringCat(pStatusText, " = Bad_CommunicationError", nStatusTextSize);
				break;
			case 0x80060000:
				BrbStringCat(pStatusText, " = Bad_EncodingError", nStatusTextSize);
				break;
			case 0x80070000:
				BrbStringCat(pStatusText, " = Bad_DecodingError", nStatusTextSize);
				break;
			case 0x80080000:
				BrbStringCat(pStatusText, " = Bad_EncodingLimitsExceeded", nStatusTextSize);
				break;
			case 0x80090000:
				BrbStringCat(pStatusText, " = Bad_UnknownResponse", nStatusTextSize);
				break;
			case 0x800A0000:
				BrbStringCat(pStatusText, " = Bad_Timeout", nStatusTextSize);
				break;
			case 0x800B0000:
				BrbStringCat(pStatusText, " = Bad_ServiceUnsupported", nStatusTextSize);
				break;
			case 0x800C0000:
				BrbStringCat(pStatusText, " = Bad_Shutdown", nStatusTextSize);
				break;
			case 0x800D0000:
				BrbStringCat(pStatusText, " = Bad_ServerNotConnected", nStatusTextSize);
				break;
			case 0x800E0000:
				BrbStringCat(pStatusText, " = Bad_ServerHalted", nStatusTextSize);
				break;
			case 0x800F0000:
				BrbStringCat(pStatusText, " = Bad_NothingToDo", nStatusTextSize);
				break;
			case 0x80100000:
				BrbStringCat(pStatusText, " = Bad_TooManyOperations", nStatusTextSize);
				break;
			case 0x80110000:
				BrbStringCat(pStatusText, " = Bad_DataTypeIdUnknown", nStatusTextSize);
				break;
			case 0x80120000:
				BrbStringCat(pStatusText, " = Bad_CertificateInvalid", nStatusTextSize);
				break;
			case 0x80130000:
				BrbStringCat(pStatusText, " = Bad_SecurityChecksFailed", nStatusTextSize);
				break;
			case 0x80140000:
				BrbStringCat(pStatusText, " = Bad_CertificateTimeInvalid", nStatusTextSize);
				break;
			case 0x80150000:
				BrbStringCat(pStatusText, " = Bad_CertificateIssuerTimeInvalid", nStatusTextSize);
				break;
			case 0x80160000:
				BrbStringCat(pStatusText, " = Bad_CertificateHostNameInvalid", nStatusTextSize);
				break;
			case 0x80170000:
				BrbStringCat(pStatusText, " = Bad_CertificateUriInvalid", nStatusTextSize);
				break;
			case 0x80180000:
				BrbStringCat(pStatusText, " = Bad_CertificateUseNotAllowed", nStatusTextSize);
				break;
			case 0x80190000:
				BrbStringCat(pStatusText, " = Bad_CertificateIssuerUseNotAllowed", nStatusTextSize);
				break;
			case 0x801A0000:
				BrbStringCat(pStatusText, " = Bad_CertificateUntrusted", nStatusTextSize);
				break;
			case 0x801B0000:
				BrbStringCat(pStatusText, " = Bad_CertificateRevocationUnknown", nStatusTextSize);
				break;
			case 0x801C0000:
				BrbStringCat(pStatusText, " = Bad_CertificateIssuerRevocationUnknown", nStatusTextSize);
				break;
			case 0x801D0000:
				BrbStringCat(pStatusText, " = Bad_CertificateRevoked", nStatusTextSize);
				break;
			case 0x801E0000:
				BrbStringCat(pStatusText, " = Bad_CertificateIssuerRevoked", nStatusTextSize);
				break;
			case 0x801F0000:
				BrbStringCat(pStatusText, " = Bad_UserAccessDenied", nStatusTextSize);
				break;
			case 0x80200000:
				BrbStringCat(pStatusText, " = Bad_IdentityTokenInvalid", nStatusTextSize);
				break;
			case 0x80210000:
				BrbStringCat(pStatusText, " = Bad_IdentityTokenRejected", nStatusTextSize);
				break;
			case 0x80220000:
				BrbStringCat(pStatusText, " = Bad_SecureChannelIdInvalid", nStatusTextSize);
				break;
			case 0x80230000:
				BrbStringCat(pStatusText, " = Bad_InvalidTimestamp", nStatusTextSize);
				break;
			case 0x80240000:
				BrbStringCat(pStatusText, " = Bad_NonceInvalid", nStatusTextSize);
				break;
			case 0x80250000:
				BrbStringCat(pStatusText, " = Bad_SessionIdInvalid", nStatusTextSize);
				break;
			case 0x80260000:
				BrbStringCat(pStatusText, " = Bad_SessionClosed", nStatusTextSize);
				break;
			case 0x80270000:
				BrbStringCat(pStatusText, " = Bad_SessionNotActivated", nStatusTextSize);
				break;
			case 0x80280000:
				BrbStringCat(pStatusText, " = Bad_SubscriptionIdInvalid", nStatusTextSize);
				break;
			case 0x802A0000:
				BrbStringCat(pStatusText, " = Bad_RequestHeaderInvalid", nStatusTextSize);
				break;
			case 0x802B0000:
				BrbStringCat(pStatusText, " = Bad_TimestampsToReturnInvalid", nStatusTextSize);
				break;
			case 0x802C0000:
				BrbStringCat(pStatusText, " = Bad_RequestCancelledByClient", nStatusTextSize);
				break;
			case 0x80310000:
				BrbStringCat(pStatusText, " = Bad_NoCommunication", nStatusTextSize);
				break;
			case 0x80320000:
				BrbStringCat(pStatusText, " = Bad_WaitingForInitialData", nStatusTextSize);
				break;
			case 0x80330000:
				BrbStringCat(pStatusText, " = Bad_NodeIdInvalid", nStatusTextSize);
				break;
			case 0x80340000:
				BrbStringCat(pStatusText, " = Bad_NodeIdUnknown", nStatusTextSize);
				break;
			case 0x80350000:
				BrbStringCat(pStatusText, " = Bad_AttributeIdInvalid", nStatusTextSize);
				break;
			case 0x80360000:
				BrbStringCat(pStatusText, " = Bad_IndexRangeInvalid", nStatusTextSize);
				break;
			case 0x80370000:
				BrbStringCat(pStatusText, " = Bad_IndexRangeNoData", nStatusTextSize);
				break;
			case 0x80380000:
				BrbStringCat(pStatusText, " = Bad_DataEncodingInvalid", nStatusTextSize);
				break;
			case 0x80390000:
				BrbStringCat(pStatusText, " = Bad_DataEncodingUnsupported", nStatusTextSize);
				break;
			case 0x803A0000:
				BrbStringCat(pStatusText, " = Bad_NotReadable", nStatusTextSize);
				break;
			case 0x803B0000:
				BrbStringCat(pStatusText, " = Bad_NotWritable", nStatusTextSize);
				break;
			case 0x803C0000:
				BrbStringCat(pStatusText, " = Bad_OutOfRange", nStatusTextSize);
				break;
			case 0x803D0000:
				BrbStringCat(pStatusText, " = Bad_NotSupported", nStatusTextSize);
				break;
			case 0x803E0000:
				BrbStringCat(pStatusText, " = Bad_NotFound", nStatusTextSize);
				break;
			case 0x803F0000:
				BrbStringCat(pStatusText, " = Bad_ObjectDeleted", nStatusTextSize);
				break;
			case 0x80400000:
				BrbStringCat(pStatusText, " = Bad_NotImplemented", nStatusTextSize);
				break;
			case 0x80410000:
				BrbStringCat(pStatusText, " = Bad_MonitoringModeInvalid", nStatusTextSize);
				break;
			case 0x80420000:
				BrbStringCat(pStatusText, " = Bad_MonitoredItemIdInvalid", nStatusTextSize);
				break;
			case 0x80430000:
				BrbStringCat(pStatusText, " = Bad_MonitoredItemFilterInvalid", nStatusTextSize);
				break;
			case 0x80440000:
				BrbStringCat(pStatusText, " = Bad_MonitoredItemFilterUnsupported", nStatusTextSize);
				break;
			case 0x80450000:
				BrbStringCat(pStatusText, " = Bad_FilterNotAllowed", nStatusTextSize);
				break;
			case 0x80460000:
				BrbStringCat(pStatusText, " = Bad_StructureMissing", nStatusTextSize);
				break;
			case 0x80470000:
				BrbStringCat(pStatusText, " = Bad_EventFilterInvalid", nStatusTextSize);
				break;
			case 0x80480000:
				BrbStringCat(pStatusText, " = Bad_ContentFilterInvalid", nStatusTextSize);
				break;
			case 0x80490000:
				BrbStringCat(pStatusText, " = Bad_FilterOperandInvalid", nStatusTextSize);
				break;
			case 0x804A0000:
				BrbStringCat(pStatusText, " = Bad_ContinuationPointInvalid", nStatusTextSize);
				break;
			case 0x804B0000:
				BrbStringCat(pStatusText, " = Bad_NoContinuationPoints", nStatusTextSize);
				break;
			case 0x804C0000:
				BrbStringCat(pStatusText, " = Bad_ReferenceTypeIdInvalid", nStatusTextSize);
				break;
			case 0x804D0000:
				BrbStringCat(pStatusText, " = Bad_BrowseDirectionInvalid", nStatusTextSize);
				break;
			case 0x804E0000:
				BrbStringCat(pStatusText, " = Bad_NodeNotInView", nStatusTextSize);
				break;
			case 0x804F0000:
				BrbStringCat(pStatusText, " = Bad_ServerUriInvalid", nStatusTextSize);
				break;
			case 0x80500000:
				BrbStringCat(pStatusText, " = Bad_ServerNameMissing", nStatusTextSize);
				break;
			case 0x80510000:
				BrbStringCat(pStatusText, " = Bad_DiscoveryUrlMissing", nStatusTextSize);
				break;
			case 0x80520000:
				BrbStringCat(pStatusText, " = Bad_SempahoreFileMissing", nStatusTextSize);
				break;
			case 0x80530000:
				BrbStringCat(pStatusText, " = Bad_RequestTypeInvalid", nStatusTextSize);
				break;
			case 0x80540000:
				BrbStringCat(pStatusText, " = Bad_SecurityModeRejected", nStatusTextSize);
				break;
			case 0x80550000:
				BrbStringCat(pStatusText, " = Bad_SecurityPolicyRejected", nStatusTextSize);
				break;
			case 0x80560000:
				BrbStringCat(pStatusText, " = Bad_TooManySessions", nStatusTextSize);
				break;
			case 0x80570000:
				BrbStringCat(pStatusText, " = Bad_UserSignatureInvalid", nStatusTextSize);
				break;
			case 0x80580000:
				BrbStringCat(pStatusText, " = Bad_ApplicationSignatureInvalid", nStatusTextSize);
				break;
			case 0x80590000:
				BrbStringCat(pStatusText, " = Bad_NoValidCertificates", nStatusTextSize);
				break;
			case 0x805A0000:
				BrbStringCat(pStatusText, " = Bad_RequestCancelledByRequest", nStatusTextSize);
				break;
			case 0x805B0000:
				BrbStringCat(pStatusText, " = Bad_ParentNodeIdInvalid", nStatusTextSize);
				break;
			case 0x805C0000:
				BrbStringCat(pStatusText, " = Bad_ReferenceNotAllowed", nStatusTextSize);
				break;
			case 0x805D0000:
				BrbStringCat(pStatusText, " = Bad_NodeIdRejected", nStatusTextSize);
				break;
			case 0x805E0000:
				BrbStringCat(pStatusText, " = Bad_NodeIdExists", nStatusTextSize);
				break;
			case 0x805F0000:
				BrbStringCat(pStatusText, " = Bad_NodeClassInvalid", nStatusTextSize);
				break;
			case 0x80600000:
				BrbStringCat(pStatusText, " = Bad_BrowseNameInvalid", nStatusTextSize);
				break;
			case 0x80610000:
				BrbStringCat(pStatusText, " = Bad_BrowseNameDuplicated", nStatusTextSize);
				break;
			case 0x80620000:
				BrbStringCat(pStatusText, " = Bad_NodeAttributesInvalid", nStatusTextSize);
				break;
			case 0x80630000:
				BrbStringCat(pStatusText, " = Bad_TypeDefinitionInvalid", nStatusTextSize);
				break;
			case 0x80640000:
				BrbStringCat(pStatusText, " = Bad_SourceNodeIdInvalid", nStatusTextSize);
				break;
			case 0x80650000:
				BrbStringCat(pStatusText, " = Bad_TargetNodeIdInvalid", nStatusTextSize);
				break;
			case 0x80660000:
				BrbStringCat(pStatusText, " = Bad_DuplicateReferenceNotAllowed", nStatusTextSize);
				break;
			case 0x80670000:
				BrbStringCat(pStatusText, " = Bad_InvalidSelfReference", nStatusTextSize);
				break;
			case 0x80680000:
				BrbStringCat(pStatusText, " = Bad_ReferenceLocalOnly", nStatusTextSize);
				break;
			case 0x80690000:
				BrbStringCat(pStatusText, " = Bad_NoDeleteRights", nStatusTextSize);
				break;
			case 0x806A0000:
				BrbStringCat(pStatusText, " = Bad_ServerIndexInvalid", nStatusTextSize);
				break;
			case 0x806B0000:
				BrbStringCat(pStatusText, " = Bad_ViewIdUnknown", nStatusTextSize);
				break;
			case 0x806D0000:
				BrbStringCat(pStatusText, " = Bad_TooManyMatches", nStatusTextSize);
				break;
			case 0x806E0000:
				BrbStringCat(pStatusText, " = Bad_QueryTooComplex", nStatusTextSize);
				break;
			case 0x806F0000:
				BrbStringCat(pStatusText, " = Bad_NoMatch", nStatusTextSize);
				break;
			case 0x80700000:
				BrbStringCat(pStatusText, " = Bad_MaxAgeInvalid", nStatusTextSize);
				break;
			case 0x80710000:
				BrbStringCat(pStatusText, " = Bad_HistoryOperationInvalid", nStatusTextSize);
				break;
			case 0x80720000:
				BrbStringCat(pStatusText, " = Bad_HistoryOperationUnsupported", nStatusTextSize);
				break;
			case 0x80730000:
				BrbStringCat(pStatusText, " = Bad_WriteNotSupported", nStatusTextSize);
				break;
			case 0x80740000:
				BrbStringCat(pStatusText, " = Bad_TypeMismatch", nStatusTextSize);
				break;
			case 0x80750000:
				BrbStringCat(pStatusText, " = Bad_MethodInvalid", nStatusTextSize);
				break;
			case 0x80760000:
				BrbStringCat(pStatusText, " = Bad_ArgumentsMissing", nStatusTextSize);
				break;
			case 0x80770000:
				BrbStringCat(pStatusText, " = Bad_TooManySubscriptions", nStatusTextSize);
				break;
			case 0x80780000:
				BrbStringCat(pStatusText, " = Bad_TooManyPublishRequests", nStatusTextSize);
				break;
			case 0x80790000:
				BrbStringCat(pStatusText, " = Bad_NoSubscription", nStatusTextSize);
				break;
			case 0x807A0000:
				BrbStringCat(pStatusText, " = Bad_SequenceNumberUnknown", nStatusTextSize);
				break;
			case 0x807B0000:
				BrbStringCat(pStatusText, " = Bad_MessageNotAvailable", nStatusTextSize);
				break;
			case 0x807C0000:
				BrbStringCat(pStatusText, " = Bad_InsufficientClientProfile", nStatusTextSize);
				break;
			case 0x807D0000:
				BrbStringCat(pStatusText, " = Bad_TcpServerTooBusy", nStatusTextSize);
				break;
			case 0x807E0000:
				BrbStringCat(pStatusText, " = Bad_TcpMessageTypeInvalid", nStatusTextSize);
				break;
			case 0x807F0000:
				BrbStringCat(pStatusText, " = Bad_TcpSecureChannelUnknown", nStatusTextSize);
				break;
			case 0x80800000:
				BrbStringCat(pStatusText, " = Bad_TcpMessageTooLarge", nStatusTextSize);
				break;
			case 0x80810000:
				BrbStringCat(pStatusText, " = Bad_TcpNotEnoughResources", nStatusTextSize);
				break;
			case 0x80820000:
				BrbStringCat(pStatusText, " = Bad_TcpInternalError", nStatusTextSize);
				break;
			case 0x80830000:
				BrbStringCat(pStatusText, " = Bad_TcpEndpointUrlInvalid", nStatusTextSize);
				break;
			case 0x80840000:
				BrbStringCat(pStatusText, " = Bad_RequestInterrupted", nStatusTextSize);
				break;
			case 0x80850000:
				BrbStringCat(pStatusText, " = Bad_RequestTimeout", nStatusTextSize);
				break;
			case 0x80860000:
				BrbStringCat(pStatusText, " = Bad_SecureChannelClosed", nStatusTextSize);
				break;
			case 0x80870000:
				BrbStringCat(pStatusText, " = Bad_SecureChannelTokenUnknown", nStatusTextSize);
				break;
			case 0x80880000:
				BrbStringCat(pStatusText, " = Bad_SequenceNumberInvalid", nStatusTextSize);
				break;
			case 0x80890000:
				BrbStringCat(pStatusText, " = Bad_ConfigurationError", nStatusTextSize);
				break;
			case 0x808A0000:
				BrbStringCat(pStatusText, " = Bad_NotConnected", nStatusTextSize);
				break;
			case 0x808B0000:
				BrbStringCat(pStatusText, " = Bad_DeviceFailure", nStatusTextSize);
				break;
			case 0x808C0000:
				BrbStringCat(pStatusText, " = Bad_SensorFailure", nStatusTextSize);
				break;
			case 0x808D0000:
				BrbStringCat(pStatusText, " = Bad_OutOfService", nStatusTextSize);
				break;
			case 0x808E0000:
				BrbStringCat(pStatusText, " = Bad_DeadbandFilterInvalid", nStatusTextSize);
				break;
			case 0x80970000:
				BrbStringCat(pStatusText, " = Bad_RefreshInProgress", nStatusTextSize);
				break;
			case 0x80980000:
				BrbStringCat(pStatusText, " = Bad_ConditionAlreadyDisabled", nStatusTextSize);
				break;
			case 0x80990000:
				BrbStringCat(pStatusText, " = Bad_ConditionDisabled", nStatusTextSize);
				break;
			case 0x809A0000:
				BrbStringCat(pStatusText, " = Bad_EventIdUnknown", nStatusTextSize);
				break;
			case 0x809B0000:
				BrbStringCat(pStatusText, " = Bad_NoData", nStatusTextSize);
				break;
			case 0x809D0000:
				BrbStringCat(pStatusText, " = Bad_DataLost", nStatusTextSize);
				break;
			case 0x809E0000:
				BrbStringCat(pStatusText, " = Bad_DataUnavailable", nStatusTextSize);
				break;
			case 0x809F0000:
				BrbStringCat(pStatusText, " = Bad_EntryExists", nStatusTextSize);
				break;
			case 0x80A00000:
				BrbStringCat(pStatusText, " = Bad_NoEntryExists", nStatusTextSize);
				break;
			case 0x80A10000:
				BrbStringCat(pStatusText, " = Bad_TimestampNotSupported", nStatusTextSize);
				break;
			case 0x80AB0000:
				BrbStringCat(pStatusText, " = Bad_InvalidArgument", nStatusTextSize);
				break;
			case 0x80AC0000:
				BrbStringCat(pStatusText, " = Bad_ConnectionRejected", nStatusTextSize);
				break;
			case 0x80AD0000:
				BrbStringCat(pStatusText, " = Bad_Disconnect", nStatusTextSize);
				break;
			case 0x80AE0000:
				BrbStringCat(pStatusText, " = Bad_ConnectionClosed", nStatusTextSize);
				break;
			case 0x80AF0000:
				BrbStringCat(pStatusText, " = Bad_InvalidState", nStatusTextSize);
				break;
			case 0x80B00000:
				BrbStringCat(pStatusText, " = Bad_EndOfStream", nStatusTextSize);
				break;
			case 0x80B10000:
				BrbStringCat(pStatusText, " = Bad_NoDataAvailable", nStatusTextSize);
				break;
			case 0x80B20000:
				BrbStringCat(pStatusText, " = Bad_WaitingForResponse", nStatusTextSize);
				break;
			case 0x80B30000:
				BrbStringCat(pStatusText, " = Bad_OperationAbandoned", nStatusTextSize);
				break;
			case 0x80B40000:
				BrbStringCat(pStatusText, " = Bad_ExpectedStreamToBlock", nStatusTextSize);
				break;
			case 0x80B50000:
				BrbStringCat(pStatusText, " = Bad_WouldBlock", nStatusTextSize);
				break;
			case 0x80B60000:
				BrbStringCat(pStatusText, " = Bad_SyntaxError", nStatusTextSize);
				break;
			case 0x80B70000:
				BrbStringCat(pStatusText, " = Bad_MaxConnectionsReached", nStatusTextSize);
				break;
			case 0x80B80000:
				BrbStringCat(pStatusText, " = Bad_RequestTooLarge", nStatusTextSize);
				break;
			case 0x80B90000:
				BrbStringCat(pStatusText, " = Bad_ResponseTooLarge", nStatusTextSize);
				break;
			case 0x80BB0000:
				BrbStringCat(pStatusText, " = Bad_EventNotAcknowledgeable", nStatusTextSize);
				break;
			case 0x80BD0000:
				BrbStringCat(pStatusText, " = Bad_InvalidTimestampArgument", nStatusTextSize);
				break;
			case 0x80BE0000:
				BrbStringCat(pStatusText, " = Bad_ProtocolVersionUnsupported", nStatusTextSize);
				break;
			case 0x80BF0000:
				BrbStringCat(pStatusText, " = Bad_StateNotActive", nStatusTextSize);
				break;
			case 0x80C10000:
				BrbStringCat(pStatusText, " = Bad_FilterOperatorInvalid", nStatusTextSize);
				break;
			case 0x80C20000:
				BrbStringCat(pStatusText, " = Bad_FilterOperatorUnsupported", nStatusTextSize);
				break;
			case 0x80C30000:
				BrbStringCat(pStatusText, " = Bad_FilterOperandCountMismatch", nStatusTextSize);
				break;
			case 0x80C40000:
				BrbStringCat(pStatusText, " = Bad_FilterElementInvalid", nStatusTextSize);
				break;
			case 0x80C50000:
				BrbStringCat(pStatusText, " = Bad_FilterLiteralInvalid", nStatusTextSize);
				break;
			case 0x80C60000:
				BrbStringCat(pStatusText, " = Bad_IdentityChangeNotSupported", nStatusTextSize);
				break;
			case 0x80C80000:
				BrbStringCat(pStatusText, " = Bad_NotTypeDefinition", nStatusTextSize);
				break;
			case 0x80C90000:
				BrbStringCat(pStatusText, " = Bad_ViewTimestampInvalid", nStatusTextSize);
				break;
			case 0x80CA0000:
				BrbStringCat(pStatusText, " = Bad_ViewParameterMismatch", nStatusTextSize);
				break;
			case 0x80CB0000:
				BrbStringCat(pStatusText, " = Bad_ViewVersionInvalid", nStatusTextSize);
				break;
			case 0x80CC0000:
				BrbStringCat(pStatusText, " = Bad_ConditionAlreadyEnabled", nStatusTextSize);
				break;
			case 0x80CD0000:
				BrbStringCat(pStatusText, " = Bad_DialogNotActive", nStatusTextSize);
				break;
			case 0x80CE0000:
				BrbStringCat(pStatusText, " = Bad_DialogResponseInvalid", nStatusTextSize);
				break;
			case 0x80CF0000:
				BrbStringCat(pStatusText, " = Bad_ConditionBranchAlreadyAcked", nStatusTextSize);
				break;
			case 0x80D00000:
				BrbStringCat(pStatusText, " = Bad_ConditionBranchAlreadyConfirmed", nStatusTextSize);
				break;
			case 0x80D10000:
				BrbStringCat(pStatusText, " = Bad_ConditionAlreadyShelved", nStatusTextSize);
				break;
			case 0x80D20000:
				BrbStringCat(pStatusText, " = Bad_ConditionNotShelved", nStatusTextSize);
				break;
			case 0x80D30000:
				BrbStringCat(pStatusText, " = Bad_ShelvingTimeOutOfRange", nStatusTextSize);
				break;
			case 0x80D40000:
				BrbStringCat(pStatusText, " = Bad_AggregateListMismatch", nStatusTextSize);
				break;
			case 0x80D50000:
				BrbStringCat(pStatusText, " = Bad_AggregateNotSupported", nStatusTextSize);
				break;
			case 0x80D60000:
				BrbStringCat(pStatusText, " = Bad_AggregateInvalidInputs", nStatusTextSize);
				break;
			case 0x80D70000:
				BrbStringCat(pStatusText, " = Bad_BoundNotFound", nStatusTextSize);
				break;
			case 0x80D80000:
				BrbStringCat(pStatusText, " = Bad_BoundNotSupported", nStatusTextSize);
				break;
			case 0x80DA0000:
				BrbStringCat(pStatusText, " = Bad_AggregateConfigurationRejected", nStatusTextSize);
				break;
			case 0x80DB0000:
				BrbStringCat(pStatusText, " = Bad_TooManyMonitoredItems", nStatusTextSize);
				break;

			case 0x81010000:
				BrbStringCat(pStatusText, " = Bad_SignatureInvalid", nStatusTextSize);
				break;
			case 0x81040000:
				BrbStringCat(pStatusText, " = Bad_ExtensibleParameterInvalid", nStatusTextSize);
				break;
			case 0x81050000:
				BrbStringCat(pStatusText, " = Bad_ExtensibleParameterUnsupported", nStatusTextSize);
				break;
			case 0x81060000:
				BrbStringCat(pStatusText, " = Bad_HostUnknown", nStatusTextSize);
				break;
			case 0x81070000:
				BrbStringCat(pStatusText, " = Bad_TooManyPosts", nStatusTextSize);
				break;
			case 0x81080000:
				BrbStringCat(pStatusText, " = Bad_SecurityConfig", nStatusTextSize);
				break;
			case 0x81090000:
				BrbStringCat(pStatusText, " = Bad_FileNotFound", nStatusTextSize);
				break;
			case 0x810A0000:
				BrbStringCat(pStatusText, " = Bad_FileExists", nStatusTextSize);
				break;

			case 0xA0010000:
				BrbStringCat(pStatusText, " = PlcOpen_BadFwPermanentError", nStatusTextSize);
				break;
			case 0xA0020000:
				BrbStringCat(pStatusText, " = PlcOpen_BadFwTempError", nStatusTextSize);
				break;
			case 0xA0030000:
				BrbStringCat(pStatusText, " = PlcOpen_BadConnectionError", nStatusTextSize);
				break;
			case 0xA0040000:
				BrbStringCat(pStatusText, " = PlcOpen_BadHostNotFound", nStatusTextSize);
				break;
			case 0xA0050000:
				BrbStringCat(pStatusText, " = PlcOpen_BadAlreadyConnected", nStatusTextSize);
				break;
			case 0xA0060000:
				BrbStringCat(pStatusText, " = PlcOpen_BadSecurityFailed", nStatusTextSize);
				break;
			case 0xA0070000:
				BrbStringCat(pStatusText, " = PlcOpen_BadSuspended", nStatusTextSize);
				break;
			case 0xA0080000:
				BrbStringCat(pStatusText, " = PlcOpen_BadConnectionInvalidHdl", nStatusTextSize);
				break;
			case 0xA0090000:
				BrbStringCat(pStatusText, " = PlcOpen_BadNsNotFound", nStatusTextSize);
				break;
			case 0xA00A0000:
				BrbStringCat(pStatusText, " = PlcOpen_BadResultTooLong", nStatusTextSize);
				break;
			case 0xA00B0000:
				BrbStringCat(pStatusText, " = PlcOpen_BadInvalidType", nStatusTextSize);
				break;
			case 0xA00C0000:
				BrbStringCat(pStatusText, " = PlcOpen_BadNodeInvalidHdl", nStatusTextSize);
				break;
			case 0xA00D0000:
				BrbStringCat(pStatusText, " = PlcOpen_BadMethodInvalidHdl", nStatusTextSize);
				break;
			case 0xA00E0000:
				BrbStringCat(pStatusText, " = PlcOpen_BadReadFailed", nStatusTextSize);
				break;
			case 0xA00F0000:
				BrbStringCat(pStatusText, " = PlcOpen_BadWriteFailed", nStatusTextSize);
				break;
			case 0xA0100000:
				BrbStringCat(pStatusText, " = PlcOpen_BadCallFailed", nStatusTextSize);
				break;
			case 0xA0110000:
				BrbStringCat(pStatusText, " = PlcOpen_BadInParamFailed", nStatusTextSize);
				break;
			case 0xA0120000:
				BrbStringCat(pStatusText, " = PlcOpen_BadOutParamFailed", nStatusTextSize);
				break;
			case 0xA0130000:
				BrbStringCat(pStatusText, " = PlcOpen_BadSubscriptionInvalidHdl", nStatusTextSize);
				break;
			case 0xA0140000:
				BrbStringCat(pStatusText, " = PlcOpen_BadMonitoredItemInvalidHdl", nStatusTextSize);
				break;
			case 0xA0150000:
				BrbStringCat(pStatusText, " = PlcOpen_BadMonitoredItemSyncMismatch", nStatusTextSize);
				break;

			case 0xB0020000:
				BrbStringCat(pStatusText, " = PlcOpen_BadUnexpectedNoOfResults", nStatusTextSize);
				break;
			case 0xB0030000:
				BrbStringCat(pStatusText, " = PlcOpen_BadIndexOutOfRange", nStatusTextSize);
				break;
			case 0xB0040000:
				BrbStringCat(pStatusText, " = PlcOpen_BadVariableNameInvalid", nStatusTextSize);
				break;
			case 0xB0050000:
				BrbStringCat(pStatusText, " = PlcOpen_BadTypeNameInvalid", nStatusTextSize);
				break;
			case 0xB0060000:
				BrbStringCat(pStatusText, " = PlcOpen_BadBrowseNameNotFound", nStatusTextSize);
				break;
			case 0xB0070000:
				BrbStringCat(pStatusText, " = PlcOpen_BadConfigAmbiguity", nStatusTextSize);
				break;
			case 0xB0080000:
				BrbStringCat(pStatusText, " = PlcOpen_BadEventFieldSelection", nStatusTextSize);
				break;
			case 0xB0090000:
				BrbStringCat(pStatusText, " = PlcOpen_BadEventContentFilter", nStatusTextSize);
				break;
			case 0xB00C0000:
				BrbStringCat(pStatusText, " = PlcOpen_BadElementCount", nStatusTextSize);
				break;
			case 0xB00D0000:
				BrbStringCat(pStatusText, " = PlcOpen_BadMonitoringQueueSize", nStatusTextSize);
				break;
			case 0xB00E0000:
				BrbStringCat(pStatusText, " = PlcOpen_BadServerNotRunning", nStatusTextSize);
				break;
			case 0xB00F0000:
				BrbStringCat(pStatusText, " = PlcOpen_BadNodeIdAlreayUsed", nStatusTextSize);
				break;
			case 0xB0100000:
				BrbStringCat(pStatusText, " = PlcOpen_BadMethodCallHandleInvalid", nStatusTextSize);
				break;
			case 0xB0110000:
				BrbStringCat(pStatusText, " = PlcOpen_BadMethodNameInvalid", nStatusTextSize);
				break;
			case 0xB0190000:
				BrbStringCat(pStatusText, " = PlcOpen_BadInvalidEventFieldValue", nStatusTextSize);
				break;

			case 0xB00B0000:
				BrbStringCat(pStatusText, " = Bad_InvalidNodeCount", nStatusTextSize);
				break;
			case 0xB0120000:
				BrbStringCat(pStatusText, " = Bad_NoAuthorization", nStatusTextSize);
				break;
			case 0xB0130000:
				BrbStringCat(pStatusText, " = Bad_UnknownRole", nStatusTextSize);
				break;
			case 0xB0140000:
				BrbStringCat(pStatusText, " = Bad_UnknownAccessRight", nStatusTextSize);
				break;
			case 0xB0150000:
				BrbStringCat(pStatusText, " = Bad_NoRoles", nStatusTextSize);
				break;
			case 0xB0160000:
				BrbStringCat(pStatusText, " = Bad_TooManyRoles", nStatusTextSize);
				break;
			case 0xB0170000:
				BrbStringCat(pStatusText, " = Bad_DuplicateRole", nStatusTextSize);
				break;
			case 0xB0180000:
				BrbStringCat(pStatusText, " = Bad_InvisibleNode", nStatusTextSize);
				break;

			default:
				nStatus = 0x803D0000; // Bad_NotSupported
				break;

		}
	}
	return nStatus;
}

// NOLINTEND(readability-*, bugprone-easily-swappable-parameters, bugprone-branch-clone, clang-diagnostic-invalid-utf8, clang-diagnostic-invalid-source-encoding, clang-diagnostic-pointer-arith, clang-diagnostic-strict-prototypes, hicpp-uppercase-literal-suffix, cppcoreguidelines-*, performance-*)
```

#### Package Logical/Libraries/BrbLibUa/General/Nodes - Funktionen für OpcUa-Knoten

#### BrbUaSetNodeId.c
```c
#include <bur/plctypes.h>
#ifdef __cplusplus
	extern "C"
	{
#endif

#include "BrbLibUa.h"
#include <string.h>

#ifdef __cplusplus
	};
#endif

// NOLINTBEGIN(readability-*, bugprone-easily-swappable-parameters, bugprone-branch-clone, clang-diagnostic-invalid-utf8, clang-diagnostic-invalid-source-encoding, clang-diagnostic-pointer-arith, clang-diagnostic-strict-prototypes, hicpp-uppercase-literal-suffix, cppcoreguidelines-*, performance-*)

/* Besetzt eine textuelle NodeId */
plcdword BrbUaSetNodeId(struct UANodeID* pNodeId, plcstring* sIdentifier, unsigned short nNamespaceIndex)
{
	DWORD nStatus = 0x80460000; // = Bad_StructureMissing
	if(pNodeId != 0)
	{
		nStatus = 0x00000000; // = Good
		BrbStringCopy(pNodeId->Identifier, sIdentifier, sizeof(pNodeId->Identifier));
		pNodeId->NamespaceIndex = nNamespaceIndex;
		if(BrbStringIsNumerical(sIdentifier) == 1)
		{
			pNodeId->IdentifierType = UAIdentifierType_Numeric;
		}
		else
		{
			pNodeId->IdentifierType = UAIdentifierType_String;
		}
	}
	return nStatus;
}

// NOLINTEND(readability-*, bugprone-easily-swappable-parameters, bugprone-branch-clone, clang-diagnostic-invalid-utf8, clang-diagnostic-invalid-source-encoding, clang-diagnostic-pointer-arith, clang-diagnostic-strict-prototypes, hicpp-uppercase-literal-suffix, cppcoreguidelines-*, performance-*)
```

#### BrbUaSetNodeIdNum.c
```c
#include <bur/plctypes.h>
#ifdef __cplusplus
	extern "C"
	{
#endif

#include "BrbLibUa.h"
#include <string.h>

#ifdef __cplusplus
	};
#endif

// NOLINTBEGIN(readability-*, bugprone-easily-swappable-parameters, bugprone-branch-clone, clang-diagnostic-invalid-utf8, clang-diagnostic-invalid-source-encoding, clang-diagnostic-pointer-arith, clang-diagnostic-strict-prototypes, hicpp-uppercase-literal-suffix, cppcoreguidelines-*, performance-*)

/* Besetzt eine numerische NodeId */
plcdword BrbUaSetNodeIdNum(struct UANodeID* pNodeId, unsigned long nIdentifier, unsigned short nNamespaceIndex)
{
	DWORD nStatus = 0x80460000; // = Bad_StructureMissing
	if(pNodeId != 0)
	{
		nStatus = 0x00000000; // = Good
		BrbUdintToAscii(nIdentifier, pNodeId->Identifier);
		pNodeId->NamespaceIndex = nNamespaceIndex;
		pNodeId->IdentifierType = UAIdentifierType_Numeric;
	}
	return nStatus;
}

// NOLINTEND(readability-*, bugprone-easily-swappable-parameters, bugprone-branch-clone, clang-diagnostic-invalid-utf8, clang-diagnostic-invalid-source-encoding, clang-diagnostic-pointer-arith, clang-diagnostic-strict-prototypes, hicpp-uppercase-literal-suffix, cppcoreguidelines-*, performance-*)
```

#### BrbUaGetRandomNodeId.c
```c
#include <bur/plctypes.h>
#ifdef __cplusplus
	extern "C"
	{
#endif

#include "BrbLibUa.h"
#include <AnsiCFunc.h>
#include <string.h>

#ifdef __cplusplus
	};
#endif

// NOLINTBEGIN(readability-*, bugprone-easily-swappable-parameters, bugprone-branch-clone, clang-diagnostic-invalid-utf8, clang-diagnostic-invalid-source-encoding, clang-diagnostic-pointer-arith, clang-diagnostic-strict-prototypes, hicpp-uppercase-literal-suffix, cppcoreguidelines-*, performance-*)

/* Erzeugt eine zufällige NodeId */
plcdword BrbUaGetRandomNodeId(struct UANodeID* pNodeId, enum UAIdentifierType eIdentifierType)
{
	DWORD nStatus = 0x80460000; // = Bad_StructureMissing
	if(pNodeId != 0)
	{
		nStatus = 0x00000000; // = Good
		UINT nNamespaceIndex = (UINT)BrbGetRandomDint(0, 10);
		if(eIdentifierType == UAIdentifierType_String)
		{
			pNodeId->IdentifierType = UAIdentifierType_String;
			pNodeId->NamespaceIndex = nNamespaceIndex;
			BrbGetRandomString(pNodeId->Identifier, sizeof(pNodeId->Identifier), 20, eBRB_RANDOM_STRING_UPPER_LETTERS + eBRB_RANDOM_STRING_LOWER_LETTERS); // NOLINT(clang-diagnostic-assign-enum)
		}
		else if(eIdentifierType == UAIdentifierType_GUID)
		{
			pNodeId->IdentifierType = UAIdentifierType_GUID;
			pNodeId->NamespaceIndex = nNamespaceIndex;
			BrbUaGetRandomGuidString((BrUaGuidString*)&pNodeId->Identifier, sizeof(pNodeId->Identifier), 1);
		}
		else if(eIdentifierType == UAIdentifierType_Opaque)
		{
			pNodeId->IdentifierType = UAIdentifierType_Opaque;
			pNodeId->NamespaceIndex = nNamespaceIndex;
			BrbStringCopy((STRING*)&pNodeId->Identifier, "", sizeof(pNodeId->Identifier));
			nStatus = 0x803D0000; // = Bad_NotSupported
		}
		else
		{
			pNodeId->IdentifierType = UAIdentifierType_Numeric;
			DINT nType = BrbGetRandomDint(0,2);
			if(nType == 0)
			{
				// 2 Byte
				pNodeId->NamespaceIndex = 0;
				UDINT nIdentifier = (UDINT)BrbGetRandomUdint(0,255);
				BrbUdintToAscii(nIdentifier, pNodeId->Identifier);
			}
			else if(nType == 1)
			{
				// 4 Byte
				pNodeId->NamespaceIndex = nNamespaceIndex;
				UDINT nIdentifier = (UINT)BrbGetRandomDint(4096, 65535);
				BrbUdintToAscii(nIdentifier, pNodeId->Identifier);
			}
			else
			{
				// 8 Byte
				pNodeId->NamespaceIndex = nNamespaceIndex;
				UDINT nIdentifier = BrbGetRandomUdint(65535, 4294967295UL);
				BrbUdintToAscii(nIdentifier, pNodeId->Identifier);
			}
		}
	}
	return nStatus;
}

// NOLINTEND(readability-*, bugprone-easily-swappable-parameters, bugprone-branch-clone, clang-diagnostic-invalid-utf8, clang-diagnostic-invalid-source-encoding, clang-diagnostic-pointer-arith, clang-diagnostic-strict-prototypes, hicpp-uppercase-literal-suffix, cppcoreguidelines-*, performance-*)
```

#### BrbUaAreNodeIdsEqual.c
```c
#include <bur/plctypes.h>
#ifdef __cplusplus
	extern "C"
	{
#endif

#include "BrbLibUa.h"
#include <string.h>

#ifdef __cplusplus
	};
#endif

// NOLINTBEGIN(readability-*, bugprone-easily-swappable-parameters, bugprone-branch-clone, clang-diagnostic-invalid-utf8, clang-diagnostic-invalid-source-encoding, clang-diagnostic-pointer-arith, clang-diagnostic-strict-prototypes, hicpp-uppercase-literal-suffix, cppcoreguidelines-*, performance-*)

/* Gibt zurück, ob zwei NodeIds gleich sind */
plcbit BrbUaAreNodeIdsEqual(struct UANodeID* pNodeId1, struct UANodeID* pNodeId2)
{
	if(pNodeId1 == 0)
	{
		return 0;
	}
	if(pNodeId2 == 0)
	{
		return 0;
	}
	return (memcmp(pNodeId1, pNodeId2, sizeof(UANodeID)) == 0); // NOLINT(bugprone-suspicious-memory-comparison,cert-exp42-c,cert-flp37-c)
}

// NOLINTEND(readability-*, bugprone-easily-swappable-parameters, bugprone-branch-clone, clang-diagnostic-invalid-utf8, clang-diagnostic-invalid-source-encoding, clang-diagnostic-pointer-arith, clang-diagnostic-strict-prototypes, hicpp-uppercase-literal-suffix, cppcoreguidelines-*, performance-*)
```

#### BrbUaAddNodeIdText.c - Gibt den Text einer NodeId zurück
```c
#include <bur/plctypes.h>
#ifdef __cplusplus
	extern "C"
	{
#endif

#include "BrbLibUa.h"
#include <string.h>

#ifdef __cplusplus
	};
#endif

// NOLINTBEGIN(readability-*, bugprone-easily-swappable-parameters, bugprone-branch-clone, clang-diagnostic-invalid-utf8, clang-diagnostic-invalid-source-encoding, clang-diagnostic-pointer-arith, clang-diagnostic-strict-prototypes, hicpp-uppercase-literal-suffix, cppcoreguidelines-*, performance-*)

/* Hängt den Text einer NodeId an */
plcdword BrbUaAddNodeIdText(struct UANodeID* pNodeId, plcstring* pText, unsigned long nTextSize)
{
	DWORD nStatus = 0x80460000; // = Bad_StructureMissing
	if(pNodeId != 0 && pText != 0)
	{
		nStatus = 0x00000000; // = Good
		STRING sHelp[nBRBUA_VALUE_TEXT_CHAR_MAX];
		BrbStringCat(pText, "ns=", nTextSize);
		brsitoa((DINT)pNodeId->NamespaceIndex, (UDINT)&sHelp);
		BrbStringCat(pText, sHelp, nTextSize);
		if(pNodeId->IdentifierType == UAIdentifierType_Numeric)
		{
			BrbStringCat(pText, ";i=", nTextSize);
		}
		else if(pNodeId->IdentifierType == UAIdentifierType_String)
		{
			BrbStringCat(pText, ";s=", nTextSize);
		}
		else if(pNodeId->IdentifierType == UAIdentifierType_GUID)
		{
			BrbStringCat(pText, ";g=", nTextSize);
		}
		else if(pNodeId->IdentifierType == UAIdentifierType_Opaque)
		{
			BrbStringCat(pText, ";o=", nTextSize);
		}
		else
		{
			BrbStringCat(pText, ";?=", nTextSize);
		}
		BrbStringCat(pText, pNodeId->Identifier, nTextSize);
	}
	return nStatus;
}

// NOLINTEND(readability-*, bugprone-easily-swappable-parameters, bugprone-branch-clone, clang-diagnostic-invalid-utf8, clang-diagnostic-invalid-source-encoding, clang-diagnostic-pointer-arith, clang-diagnostic-strict-prototypes, hicpp-uppercase-literal-suffix, cppcoreguidelines-*, performance-*)
```

#### BrbUaGetAttributeIdDatatype.c - Gibt den OpcUa-Datentyp für ein Attribut zurück
```c
#include <bur/plctypes.h>
#ifdef __cplusplus
	extern "C"
	{
#endif

#include "BrbLibUa.h"

#ifdef __cplusplus
	};
#endif

// NOLINTBEGIN(readability-*, bugprone-easily-swappable-parameters, bugprone-branch-clone, clang-diagnostic-invalid-utf8, clang-diagnostic-invalid-source-encoding, clang-diagnostic-pointer-arith, clang-diagnostic-strict-prototypes, hicpp-uppercase-literal-suffix, cppcoreguidelines-*, performance-*)

/* Gibt den OpcUa-Datentyp für ein Attribut zurück */
enum UAVariantType BrbUaGetAttributeIdDatatype(enum UAAttributeId eAttributeId)
{
	UAVariantType eResult = UAVariantType_Null;
	// NOLINTBEGIN(bugprone-branch-clone)
	switch(eAttributeId) // NOLINT(hicpp-multiway-paths-covered)
	{
		case UAAI_Default:
			eResult = UAVariantType_Null;
			break;
		case UAAI_NodeId:
			eResult = UAVariantType_NodeId;
			break;
		case UAAI_NodeClass:
			eResult = UAVariantType_Int32;
			break;
		case UAAI_BrowseName:
			eResult = UAVariantType_QualifiedName;
			break;
		case UAAI_DisplayName:
			eResult = UAVariantType_LocalizedText;
			break;
		case UAAI_Description:
			eResult = UAVariantType_LocalizedText;
			break;
		case UAAI_WriteMask:
			eResult = UAVariantType_UInt32;
			break;
		case UAAI_UserWriteMask:
			eResult = UAVariantType_UInt32;
			break;
		case UAAI_IsAbstract:
			eResult = UAVariantType_Boolean;
			break;
		case UAAI_Symmetric:
			eResult = UAVariantType_Boolean;
			break;
		case UAAI_InverseName:
			eResult = UAVariantType_LocalizedText;
			break;
		case UAAI_ContainsNoLoops:
			eResult = UAVariantType_Boolean;
			break;
		case UAAI_EventNotifier:
			eResult = UAVariantType_Byte;
			break;
		case UAAI_Value:
			eResult = UAVariantType_Null;
			break;
		case UAAI_DataType:
			eResult = UAVariantType_NodeId;
			break;
		case UAAI_ValueRank:
			eResult = UAVariantType_Int32;
			break;
		case UAAI_ArrayDimensions:
			break;
		case UAAI_AccessLevel:
			eResult = UAVariantType_Byte;
			break;
		case UAAI_UserAccessLevel:
			eResult = UAVariantType_Byte;
			break;
		case UAAI_MinimumSamplingInterval:
			eResult = UAVariantType_Double;
			break;
		case UAAI_Historizing:
			eResult = UAVariantType_Boolean;
			break;
		case UAAI_Executable:
			eResult = UAVariantType_Boolean;
			break;
		case UAAI_UserExecutable:
			eResult = UAVariantType_Boolean;
			break;
	}
	// NOLINTEND(bugprone-branch-clone)
	return eResult;
}

// NOLINTEND(readability-*, bugprone-easily-swappable-parameters, bugprone-branch-clone, clang-diagnostic-invalid-utf8, clang-diagnostic-invalid-source-encoding, clang-diagnostic-pointer-arith, clang-diagnostic-strict-prototypes, hicpp-uppercase-literal-suffix, cppcoreguidelines-*, performance-*)
```

#### BrbUaGetAttributeList.c
```c
#include <bur/plctypes.h>
#ifdef __cplusplus
	extern "C"
	{
#endif

#include "BrbLibUa.h"
#include <string.h>

#ifdef __cplusplus
	};
#endif

// NOLINTBEGIN(readability-*, bugprone-easily-swappable-parameters, bugprone-branch-clone, clang-diagnostic-invalid-utf8, clang-diagnostic-invalid-source-encoding, clang-diagnostic-pointer-arith, clang-diagnostic-strict-prototypes, hicpp-uppercase-literal-suffix, cppcoreguidelines-*, performance-*)

/* Gibt eine Liste mit Attribut-Texten zurück */
plcdword BrbUaGetAttributeList(struct UANodeInfo* pNodeInfo, struct BrbUaNodeInfoAttributes_TYP* pAttributes)
{
	DWORD nStatus = 0x80460000; // = Bad_StructureMissing
	if(pAttributes != 0)
	{
		memset(pAttributes, 0, sizeof(BrbUaNodeInfoAttributes_TYP));
		BrbStringCat(pAttributes->Attribute[UAAI_Default].sName, "Default", sizeof(pAttributes->Attribute[0].sName));
		BrbStringCat(pAttributes->Attribute[UAAI_NodeId].sName, "NodeId", sizeof(pAttributes->Attribute[0].sName));
		BrbStringCat(pAttributes->Attribute[UAAI_NodeClass].sName, "NodeClass", sizeof(pAttributes->Attribute[0].sName));
		BrbStringCat(pAttributes->Attribute[UAAI_BrowseName].sName, "BrowseName", sizeof(pAttributes->Attribute[0].sName));
		BrbStringCat(pAttributes->Attribute[UAAI_DisplayName].sName, "DisplayName", sizeof(pAttributes->Attribute[0].sName));
		BrbStringCat(pAttributes->Attribute[UAAI_Description].sName, "Description", sizeof(pAttributes->Attribute[0].sName));
		BrbStringCat(pAttributes->Attribute[UAAI_WriteMask].sName, "WriteMask", sizeof(pAttributes->Attribute[0].sName));
		BrbStringCat(pAttributes->Attribute[UAAI_UserWriteMask].sName, "UserWriteMask", sizeof(pAttributes->Attribute[0].sName));
		BrbStringCat(pAttributes->Attribute[UAAI_IsAbstract].sName, "IsAbstract", sizeof(pAttributes->Attribute[0].sName));
		BrbStringCat(pAttributes->Attribute[UAAI_Symmetric].sName, "Symmetric", sizeof(pAttributes->Attribute[0].sName));
		BrbStringCat(pAttributes->Attribute[UAAI_InverseName].sName, "InverseName", sizeof(pAttributes->Attribute[0].sName));
		BrbStringCat(pAttributes->Attribute[UAAI_ContainsNoLoops].sName, "ContainsNoLoops", sizeof(pAttributes->Attribute[0].sName));
		BrbStringCat(pAttributes->Attribute[UAAI_EventNotifier].sName, "EventNotifier", sizeof(pAttributes->Attribute[0].sName));
		BrbStringCat(pAttributes->Attribute[UAAI_Value].sName, "Value", sizeof(pAttributes->Attribute[0].sName));
		BrbStringCat(pAttributes->Attribute[UAAI_DataType].sName, "DataType", sizeof(pAttributes->Attribute[0].sName));
		BrbStringCat(pAttributes->Attribute[UAAI_ValueRank].sName, "ValueRank", sizeof(pAttributes->Attribute[0].sName));
		BrbStringCat(pAttributes->Attribute[UAAI_ArrayDimensions].sName, "ArrayDimensions", sizeof(pAttributes->Attribute[0].sName));
		BrbStringCat(pAttributes->Attribute[UAAI_AccessLevel].sName, "AccessLevel", sizeof(pAttributes->Attribute[0].sName));
		BrbStringCat(pAttributes->Attribute[UAAI_UserAccessLevel].sName, "UserAccessLevel", sizeof(pAttributes->Attribute[0].sName));
		BrbStringCat(pAttributes->Attribute[UAAI_MinimumSamplingInterval].sName, "MinimumSamplingInterval", sizeof(pAttributes->Attribute[0].sName));
		BrbStringCat(pAttributes->Attribute[UAAI_Historizing].sName, "Historizing", sizeof(pAttributes->Attribute[0].sName));
		BrbStringCat(pAttributes->Attribute[UAAI_Executable].sName, "Executable", sizeof(pAttributes->Attribute[0].sName));
		BrbStringCat(pAttributes->Attribute[UAAI_UserExecutable].sName, "UserExecutable", sizeof(pAttributes->Attribute[0].sName));
		if(pNodeInfo != 0)
		{
			STRING sHelp[nBRBUA_VALUE_TEXT_CHAR_MAX];
			// Default bleibt leer
			BrbUaAddNodeIdText(&pNodeInfo->NodeID, pAttributes->Attribute[UAAI_NodeId].sValue, sizeof(pAttributes->Attribute[UAAI_NodeId].sValue));
			BrbUaAddNodeClassText(pNodeInfo->NodeClass, pAttributes->Attribute[UAAI_NodeClass].sValue, sizeof(pAttributes->Attribute[UAAI_NodeClass].sValue));
			BrbStringCat(pAttributes->Attribute[UAAI_BrowseName].sValue, pNodeInfo->BrowseName, sizeof(pAttributes->Attribute[0].sValue));
			BrbStringCat(pAttributes->Attribute[UAAI_DisplayName].sValue, pNodeInfo->DisplayName.Text, sizeof(pAttributes->Attribute[0].sValue));
			BrbStringCat(pAttributes->Attribute[UAAI_Description].sValue, pNodeInfo->Description.Text, sizeof(pAttributes->Attribute[0].sValue));
			BrbUdintToAscii(pNodeInfo->WriteMask, pAttributes->Attribute[UAAI_WriteMask].sValue);
			BrbUdintToAscii(pNodeInfo->UserWriteMask, pAttributes->Attribute[UAAI_UserWriteMask].sValue);
			BrbUaAddBooleanText(pNodeInfo->IsAbstract, pAttributes->Attribute[UAAI_IsAbstract].sValue, sizeof(pAttributes->Attribute[UAAI_IsAbstract].sValue));
			BrbUaAddBooleanText(pNodeInfo->Symmetric, pAttributes->Attribute[UAAI_Symmetric].sValue, sizeof(pAttributes->Attribute[UAAI_Symmetric].sValue));
			BrbStringCat(pAttributes->Attribute[UAAI_InverseName].sValue, pNodeInfo->InverseName, sizeof(pAttributes->Attribute[0].sValue));
			BrbUaAddBooleanText(pNodeInfo->ContainsNoLoops, pAttributes->Attribute[UAAI_ContainsNoLoops].sValue, sizeof(pAttributes->Attribute[UAAI_ContainsNoLoops].sValue));
			BrbUaAddEventNotifierText(pNodeInfo->EventNotifier, pAttributes->Attribute[UAAI_EventNotifier].sValue, sizeof(pAttributes->Attribute[UAAI_EventNotifier].sValue));
			// Value bleibt leer
			UDINT nDatatypeId = BrbAsciiToUdint(pNodeInfo->DataType.Identifier);
			BrbUaAddDatatypeIdText(nDatatypeId, pAttributes->Attribute[UAAI_DataType].sValue, sizeof(pAttributes->Attribute[UAAI_DataType].sValue));
			brsitoa((DINT)pNodeInfo->ValueRank, (UDINT)&sHelp);
			BrbStringCat(pAttributes->Attribute[UAAI_ValueRank].sValue, sHelp, sizeof(pAttributes->Attribute[0].sValue));
			BrbUaAddArrayDimensionText((UDINT*)&pNodeInfo->ArrayDimension, pNodeInfo->ValueRank, pAttributes->Attribute[UAAI_ArrayDimensions].sValue, sizeof(pAttributes->Attribute[UAAI_ArrayDimensions].sValue));
			BrbUaAddAccessLevelText(pNodeInfo->AccessLevel, pAttributes->Attribute[UAAI_AccessLevel].sValue, sizeof(pAttributes->Attribute[UAAI_AccessLevel].sValue));
			BrbUaAddAccessLevelText(pNodeInfo->UserAccessLevel, pAttributes->Attribute[UAAI_UserAccessLevel].sValue, sizeof(pAttributes->Attribute[UAAI_UserAccessLevel].sValue));
			BrbUdintToAscii((UDINT)pNodeInfo->MinimumSamplingInterval, sHelp);
			BrbStringCat(pAttributes->Attribute[UAAI_MinimumSamplingInterval].sValue, sHelp, sizeof(pAttributes->Attribute[0].sValue));
			BrbUaAddBooleanText(pNodeInfo->Historizing, pAttributes->Attribute[UAAI_Historizing].sValue, sizeof(pAttributes->Attribute[UAAI_Historizing].sValue));
			BrbUaAddBooleanText(pNodeInfo->Executable, pAttributes->Attribute[UAAI_Executable].sValue, sizeof(pAttributes->Attribute[UAAI_Executable].sValue));
			BrbUaAddBooleanText(pNodeInfo->UserExecutable, pAttributes->Attribute[UAAI_UserExecutable].sValue, sizeof(pAttributes->Attribute[UAAI_UserExecutable].sValue));
			nStatus = 0x00000000; // = Good
		}
	}
	return nStatus;
}

// NOLINTEND(readability-*, bugprone-easily-swappable-parameters, bugprone-branch-clone, clang-diagnostic-invalid-utf8, clang-diagnostic-invalid-source-encoding, clang-diagnostic-pointer-arith, clang-diagnostic-strict-prototypes, hicpp-uppercase-literal-suffix, cppcoreguidelines-*, performance-*)
```

#### BrbUaAddBooleanText.c - Gibt den Text eines boolschen Werts zurück
```c
#include <bur/plctypes.h>
#ifdef __cplusplus
	extern "C"
	{
#endif

#include "BrbLibUa.h"
#include <string.h>

#ifdef __cplusplus
	};
#endif

// NOLINTBEGIN(readability-*, bugprone-easily-swappable-parameters, bugprone-branch-clone, clang-diagnostic-invalid-utf8, clang-diagnostic-invalid-source-encoding, clang-diagnostic-pointer-arith, clang-diagnostic-strict-prototypes, hicpp-uppercase-literal-suffix, cppcoreguidelines-*, performance-*)

/* Gibt den Text eines boolschen Werts zurück */
plcdword BrbUaAddBooleanText(plcbit bBoolean, plcstring* pText, unsigned long nTextSize)
{
	DWORD nStatus = 0x80460000; // = Bad_StructureMissing
	if(pText != 0)
	{
		nStatus = 0x00000000; // = Good
		if(bBoolean == 1)
		{
			BrbStringCat(pText, "True", nTextSize);
		}
		else
		{
			BrbStringCat(pText, "False", nTextSize);
		}
	}
	return nStatus;
}

// NOLINTEND(readability-*, bugprone-easily-swappable-parameters, bugprone-branch-clone, clang-diagnostic-invalid-utf8, clang-diagnostic-invalid-source-encoding, clang-diagnostic-pointer-arith, clang-diagnostic-strict-prototypes, hicpp-uppercase-literal-suffix, cppcoreguidelines-*, performance-*)
```
